(*Fixture*)

PROGRAM Fix108
	VAR_INPUT
		Enable_Prog: BOOL;
		Enable_Motion: BOOL;
		Discrete_In: udt_FixXX_Input_Image_20180202;
		Dry_Cycle: BOOL;
		Cell_In_Services: BOOL;
		Flash_Rate: BOOL;
		NodeLayout:udt_ECATNodeData_20221507;

	END_VAR

	VAR
(*Hardware Related Data Types*)
			(*Develop "Beckhoff Nodes"*)
			{attribute 'OPC.UA.DA':='1'}
			N00 AT %I*: udt_EP1111;
			{attribute 'OPC.UA.DA':='1'}
			N01 AT %I*: udt_EP1008_002_v2;
			{attribute 'OPC.UA.DA':='1'}
			N02 AT %I*: udt_EP1008_002_v2;
			{attribute 'OPC.UA.DA':='1'}
			N03 AT %I*: udt_EP1008_002_v2;
			{attribute 'OPC.UA.DA':='1'}
			N04 AT %I*: udt_EP1008_002_v2;
			{attribute 'OPC.UA.DA':='1'}
			N05 AT %I*: udt_EP1008_002_v2;
			{attribute 'OPC.UA.DA':='1'}
			N06 AT %I*: udt_EP1008_002_v2;
			{attribute 'OPC.UA.DA':='1'}
			N07 AT %I*: udt_EP1008_002_v2;
			{attribute 'OPC.UA.DA':='1'}
			N08 AT %I*: udt_EP1008_002_v2;
			{attribute 'OPC.UA.DA':='1'}
			N09 AT %I*: udt_EP1008_002_v2;
			{attribute 'OPC.UA.DA':='1'}
			N10 AT %I*: udt_EP1008_002_v2;
			{attribute 'OPC.UA.DA':='1'}
			N11 AT %I*: udt_EP1008_002_v2;
			{attribute 'OPC.UA.DA':='1'}
			N12 AT %I*: udt_EP1008_002_v2;
			{attribute 'OPC.UA.DA':='1'}
			N13 AT %I*: udt_EP1008_002_v2;
			{attribute 'OPC.UA.DA':='1'}
			N14 AT %I*: udt_EP1008_002_v2;
			{attribute 'OPC.UA.DA':='1'}
			N15 AT %I*: udt_EP1008_002_v2;
			{attribute 'OPC.UA.DA':='1'}
			N16 AT %I*: udt_EP1008_002_v2;
			{attribute 'OPC.UA.DA':='1'}
			N17 AT %I*: udt_EP1008_002_v2;
			{attribute 'OPC.UA.DA':='1'}
			N18 AT %I*: udt_EP1008_002_v2;
			{attribute 'OPC.UA.DA':='1'}
			N19 AT %I*: udt_EP1008_002_v2;
			{attribute 'OPC.UA.DA':='1'}
			N20 AT %I*: udt_EP1008_002_v2;
			{attribute 'OPC.UA.DA':='1'}
			N21 AT %I*: udt_EP1008_002_v2;
			{attribute 'OPC.UA.DA':='1'}
			N22 AT %I*: udt_EP1008_002_v2;
			{attribute 'OPC.UA.DA':='1'}
			N100 AT %Q*: udt_SMC_EX260_ValveBank;
			{attribute 'OPC.UA.DA':='1'}
			N100_STAT AT %I*:udt_SMC_EX260_Stat;
			{attribute 'OPC.UA.DA':='1'}
			N101 AT %Q*: udt_SMC_EX260_ValveBank;
			{attribute 'OPC.UA.DA':='1'}
			N101_STAT AT %I*:udt_SMC_EX260_Stat;
			{attribute 'OPC.UA.DA':='1'}
			N102 AT %Q*: udt_SMC_EX260_ValveBank;
			{attribute 'OPC.UA.DA':='1'}
			N102_STAT AT %I*:udt_SMC_EX260_Stat;

(* Nodes States*)
		NodeState: ARRAY[0..63] OF UINT;
		DiscreteNode_OK: BOOL;
(*Cable Break States*)
		ECatSlave_Cable_Breaks: ARRAY[0..1] OF DINT;
(*Standard Internal Variables*)
		(*Generic Sensor Variables*)
		All_Sensors_On: UINT;
		All_Sensors_Off: BOOL;
		All_Sensors_Off1: BOOL;
		All_Sensors_Off2: BOOL;
		(*Generic Position Variables*)
		Tool_At_Home: BOOL;
		Tool_At_Load: UINT;
		Tool_At_Weld: UINT;
		Tool_At_Rotate: UINT;
		Tool_At_Seal: UINT;
		Tool_At_Stud: UINT;
		Tool_At_Unload: UINT ;
		(*Grouping Of Items*)
		All_QAChecks_OK: BOOL;
		QAChecks_Failed: BOOL;
		(*General Internals*)
		In_Auto: BOOL;
		In_Manual: BOOL;

		Auto_Run: BOOL;
		Reset_All_Completes:BOOL;
		Load_Robots_Clear1: BOOL;
		Load_Robots_Clear2: BOOL;
		Load_Robots_Clear: BOOL;
		Load_Robots_WorkingOK1: BOOL;
		Load_Robots_WorkingOK2: BOOL;
		Load_Robots_Complete1: BOOL;
		Load_Robots_Complete2: BOOL;
		Load_Robots_PartInEOAT1: BOOL;
		Load_Robots_PartInEOAT2: BOOL;
		Load_Robots_UnclampEarly1: BOOL;
		Load_Robots_UnclampEarly2: BOOL;
		Seal_Robots_Clear: BOOL;
		Seal_Robots_WorkingOK: BOOL;
		Seal_Robots_UnclampEarly: BOOL;
		Seal_Robots_Complete: BOOL;
		Stud_Robots_Clear: BOOL;
		Stud_Robots_WorkingOK: BOOL;
		Stud_Robots_UnclampEarly: BOOL;
		Stud_Robots_Complete: BOOL;
		Weld_Robots_Clear: BOOL;
		Weld_Robots_WorkingOK: BOOL;
		Weld_Robots_UnclampEarly: BOOL;
		Weld_Robots_Complete: BOOL;
		Mig_Robots_Ready :BOOL;
		TurntableA_Clear: BOOL;
		TurntableB_Clear: BOOL;
		Turntable_Clear:BOOL;
		Turntable_WorkingOK: BOOL;
		TurntableA_Complete: BOOL;
		TurntableB_Complete: BOOL;
		Unload_Robots_Clear1: BOOL;
		Unload_Robots_WorkingOK1: BOOL;
		Unload_Robots_Complete1: BOOL;
		Unload_Robots_EOATEmpty1: BOOL;
		Unload_Robots_Clear2: BOOL;
		Unload_Robots_WorkingOK2: BOOL;
		Unload_Robots_Complete2: BOOL;
		Unload_Robots_EOATEmpty2: BOOL;
		Unload_Robots_Clear: BOOL;
		All_Robots_Clear: BOOL;

		Unload_Robot_Complete: BOOL;

		Start_Load_Robots1: BOOL;
		Start_Load_Robots2: BOOL;
		Start_Weld_Robots: BOOL;
		Start_Unload_Robots1: BOOL;
		Start_Unload_Robots2: BOOL;
		Start_Seal_Robots: BOOL;
		Start_Stud_Robots: BOOL;
		Start_TurntableA: BOOL;
		Start_TurntableB: BOOL;
		Load_Robots_Proceed1: BOOL;
		Load_Robots_Proceed2: BOOL;
		Weld_Robots_Proceed: BOOL;
		Seal_Robots_Proceed: BOOL;
		Stud_Robots_Proceed: BOOL;
		Unload_Robots_Proceed1: BOOL;
		Unload_Robots_Proceed2: BOOL;

		Prod_Inc: R_TRIG;
		Cycle_Time: TON;
		Cycle_Time_Pulse: R_TRIG;
		Load_Time: TON;
		Weld_Time: TON;
		Seal_Time: TON;
		Stud_Time: TON;
		Turn_Time: TON;
		Unload_Time: TON;
		Date_Stamp_TMR: TON;
		Date_StampHome_TMR: TON;
		CLFaulted: UDINT;
		PPFaulted: UDINT;
		Manual_Ind_HomePrompt: BOOL;
		Fixture_Allow_Model_Change: BOOL;

(*Non-Standard Variables*)

		(*FB Instances*)
		Clamp1FB: FB_Cylinder_Status;
		Clamp2FB: FB_Cylinder_Status;
		Clamp3FB: FB_Cylinder_Status;
		Clamp4FB: FB_Cylinder_Status;
		Clamp5FB: FB_Cylinder_Status;
		Clamp6FB: FB_Cylinder_Status;
		Clamp7FB: FB_Cylinder_Status;
		Clamp8FB: FB_Cylinder_Status;
		Clamp9FB: FB_Cylinder_Status;
		Clamp10FB: FB_Cylinder_Status;
		Clamp11FB: FB_Cylinder_Status;
		Clamp12FB: FB_Cylinder_Status;
		Clamp13FB: FB_Cylinder_Status;
		Clamp14FB: FB_Cylinder_Status;
		Clamp15FB: FB_Cylinder_Status;
		Clamp16FB: FB_Cylinder_Status;
		Clamp17FB: FB_Cylinder_Status;
		Clamp18FB: FB_Cylinder_Status;
		Clamp19FB: FB_Cylinder_Status;
		Clamp20FB: FB_Cylinder_Status;
		Clamp21FB: FB_Cylinder_Status;
		Clamp22FB: FB_Cylinder_Status;
		Clamp23FB: FB_Cylinder_Status;
		Clamp24FB: FB_Cylinder_Status;
		Cyl1FB: FB_TripleCylinder_20150625;
		Pin1FB: FB_Cylinder_Status;
		Pin2FB: FB_Cylinder_Status;
		Pin3FB: FB_Cylinder_Status;
		Pin4FB: FB_Cylinder_Status;
		Pin5FB: FB_Cylinder_Status;
		Pin6FB: FB_Cylinder_Status;
		Pin7FB: FB_Cylinder_Status;
		Pin8FB: FB_Cylinder_Status;
		Pin9FB: FB_Cylinder_Status;
		Pin10FB: FB_Cylinder_Status;
		Pin11FB: FB_Cylinder_Status;
		Pin12FB: FB_Cylinder_Status;
		Pin13FB: FB_Cylinder_Status;
		Pin14FB: FB_Cylinder_Status;
		Slide1FB: FB_Cylinder_Status;
		Slide2FB: FB_Cylinder_Status;
		Slide3FB: FB_Cylinder_Status;
		Slide4FB: FB_Cylinder_Status;
		Slide5FB: FB_Cylinder_Status;
		Slide6FB: FB_Cylinder_Status;
		Swing1FB: FB_Cylinder_Status;
		Swing2FB: FB_Cylinder_Status;
		Swing3FB: FB_Cylinder_Status;
		Swing4FB: FB_Cylinder_Status;
		Swing5FB: FB_Cylinder_Status;
		Swing6FB: FB_Cylinder_Status;
		QACheck1FB: FB_Cylinder_Status;
		QACheck2FB: FB_Cylinder_Status;
		CheckQA1FB: FB_GTAC_QAcheck_20150529;
		Part_Present1FB: FB_PP_Sensor;
		Part_Present2FB: FB_PP_Sensor;
		Part_Present3FB: FB_PP_Sensor;
		Part_Present4FB: FB_PP_Sensor;
		Part_Present5FB: FB_PP_Sensor;
		Part_Present6FB: FB_PP_Sensor;
		Part_Present7FB: FB_PP_Sensor;
		Part_Present8FB: FB_PP_Sensor;
		Part_Present9FB: FB_PP_Sensor;
		Part_Present10FB: FB_PP_Sensor;
		Part_Present11FB: FB_PP_Sensor;
		Part_Present12FB: FB_PP_Sensor;
		Part_Present13FB: FB_PP_Sensor;
		Part_Present14FB: FB_PP_Sensor;
		Part_Present15FB: FB_PP_Sensor;
		Part_Present16FB: FB_PP_Sensor;
		Part_Present17FB: FB_PP_Sensor;
		Part_Present18FB: FB_PP_Sensor;
		Part_Present19FB: FB_PP_Sensor;
		Part_Present20FB: FB_PP_Sensor;
		Part_Present21FB: FB_PP_Sensor;
		Part_Present22FB: FB_PP_Sensor;
		Part_Present23FB: FB_PP_Sensor;
		Part_Present24FB: FB_PP_Sensor;
		Part_Present25FB: FB_PP_Sensor;
		Part_Present26FB: FB_PP_Sensor;
		Part_Present27FB: FB_PP_Sensor;
		Part_Present28FB: FB_PP_Sensor;
		Part_Present29FB: FB_PP_Sensor;
		Part_Present30FB: FB_PP_Sensor;
		Part_Present31FB: FB_PP_Sensor;
		Part_Present32FB: FB_PP_Sensor;
		Part_Present33FB: FB_PP_Sensor;
		Part_Present34FB: FB_PP_Sensor;
		Part_Present35FB: FB_PP_Sensor;
		Part_Present36FB: FB_PP_Sensor;
		Part_Present37FB: FB_PP_Sensor;
		Part_Present38FB: FB_PP_Sensor;
		Part_Present39FB: FB_PP_Sensor;
		Part_Present40FB: FB_PP_Sensor;
		Tape_Present1FB: FB_PP_Sensor;

		(*Valve FBs*)
		Valve1FB: FB_GTAC_Valve_20170704;
		Valve2FB: FB_GTAC_Valve_20170704;
		Valve3FB: FB_GTAC_Valve_20170704;
		Valve4FB: FB_GTAC_Valve_20170704;
		Valve5FB: FB_GTAC_Valve_20170704;
		Valve6FB: FB_GTAC_Valve_20170704;
		Valve7FB: FB_GTAC_Valve_20170704;
		Valve8FB: FB_GTAC_Valve_20170704;
		Valve9FB: FB_GTAC_Valve_20170704;
		Valve10FB: FB_GTAC_Valve_20170704;
		Valve11FB: FB_GTAC_Valve_20170704;
		Valve12FB: FB_GTAC_Valve_20170704;
		Valve13FB: FB_GTAC_Valve_20170704;
		Valve14FB: FB_GTAC_Valve_20170704;
		Valve15FB: FB_GTAC_Valve_20170704;
		Valve16FB: FB_GTAC_Valve_20170704;
		Valve17FB: FB_GTAC_Valve_20170704;
		Valve18FB: FB_GTAC_Valve_20170704;
		Valve19FB: FB_GTAC_Valve_20170704;
		Valve20FB: FB_GTAC_Valve_20170704;
		Valve21FB: FB_GTAC_Valve_20170704;
		Valve22FB: FB_GTAC_Valve_20170704;
		Valve23FB: FB_GTAC_Valve_20170704;
		Valve24FB: FB_GTAC_Valve_20170704;
		Valve25FB: FB_GTAC_Valve_20170704;
		Valve26FB: FB_GTAC_Valve_20170704;
		Valve27FB: FB_GTAC_Valve_20170704;
		Valve28FB: FB_GTAC_Valve_20170704;
		Valve29FB: FB_GTAC_Valve_20170704;
		Valve30FB: FB_GTAC_Valve_20170704;
		Valve31FB: FB_GTAC_Valve_20170704;
		Valve32FB: FB_GTAC_Valve_20170704;
		Valve33FB: FB_GTAC_Valve_20170704;
		Valve34FB: FB_GTAC_Valve_20170704;
		Valve35FB: FB_GTAC_Valve_20170704;
		Valve36FB: FB_GTAC_Valve_20170704;
		Valve37FB: FB_GTAC_Valve_20170704;
		Valve38FB: FB_GTAC_Valve_20170704;
		Valve39FB: FB_GTAC_Valve_20170704;
		Valve40FB: FB_GTAC_Valve_20170704;
		Valve41FB: FB_GTAC_Valve_20170704;
		Valve42FB: FB_GTAC_Valve_20170704;
		Valve43FB: FB_GTAC_Valve_20170704;
		Valve44FB: FB_GTAC_Valve_20170704;
		Valve45FB: FB_GTAC_Valve_20170704;
		Valve46FB: FB_GTAC_Valve_20170704;
		Valve47FB: FB_GTAC_Valve_20170704;
		Valve48FB: FB_GTAC_Valve_20170704;

		(*Tool Positions*)
			(*Add User Indivdual Position Variables Here*)
			Clamp1ADVD: BOOL;
			Clamp1RETD: BOOL;
			Clamp2ADVD: BOOL;
			Clamp2RETD: BOOL;
			Clamp3ADVD: BOOL;
			Clamp3RETD: BOOL;
			Clamp4ADVD: BOOL;
			Clamp4RETD: BOOL;
			Clamp5ADVD: BOOL;
			Clamp5RETD: BOOL;
			Clamp6ADVD: BOOL;
			Clamp6RETD: BOOL;
			Clamp7ADVD: BOOL;
			Clamp7RETD: BOOL;
			Clamp8ADVD: BOOL;
			Clamp8RETD: BOOL;
			Clamp9ADVD: BOOL;
			Clamp9RETD: BOOL;
			Clamp10ADVD: BOOL;
			Clamp10RETD: BOOL;
			Clamp11ADVD: BOOL;
			Clamp11RETD: BOOL;
			Clamp12ADVD: BOOL;
			Clamp12RETD: BOOL;
			Clamp13ADVD: BOOL;
			Clamp13RETD: BOOL;
			Clamp14ADVD: BOOL;
			Clamp14RETD: BOOL;
			Clamp15ADVD: BOOL;
			Clamp15RETD: BOOL;
			Clamp16ADVD: BOOL;
			Clamp16RETD: BOOL;
			Clamp17ADVD: BOOL;
			Clamp17RETD: BOOL;
			Clamp18ADVD: BOOL;
			Clamp18RETD: BOOL;
			Clamp19ADVD: BOOL;
			Clamp19RETD: BOOL;
			Clamp20ADVD: BOOL;
			Clamp20RETD: BOOL;
			Clamp21ADVD: BOOL;
			Clamp21RETD: BOOL;
			Clamp22ADVD: BOOL;
			Clamp22RETD: BOOL;
			Clamp23ADVD: BOOL;
			Clamp23RETD: BOOL;
			Clamp24ADVD: BOOL;
			Clamp24RETD: BOOL;
			Cyl1ADVD: BOOL;
			Cyl1MID: BOOL;
			Cyl1RETD: BOOL;
			Pin1ADVD: BOOL;
			Pin1RETD: BOOL;
			Pin2ADVD: BOOL;
			Pin2RETD: BOOL;
			Pin3ADVD: BOOL;
			Pin3RETD: BOOL;
			Pin4ADVD: BOOL;
			Pin4RETD: BOOL;
			Pin5ADVD: BOOL;
			Pin5RETD: BOOL;
			Pin6ADVD: BOOL;
			Pin6RETD: BOOL;
			Pin7ADVD: BOOL;
			Pin7RETD: BOOL;
			Pin8ADVD: BOOL;
			Pin8RETD: BOOL;
			Pin9ADVD: BOOL;
			Pin9RETD: BOOL;
			Pin10ADVD: BOOL;
			Pin10RETD: BOOL;
			Pin11ADVD: BOOL;
			Pin11RETD: BOOL;
			Pin12ADVD: BOOL;
			Pin12RETD: BOOL;
			Pin13ADVD: BOOL;
			Pin13RETD: BOOL;
			Pin14ADVD: BOOL;
			Pin14RETD: BOOL;
			Slide1ADVD: BOOL;
			Slide1RETD: BOOL;
			Slide2ADVD: BOOL;
			Slide2RETD: BOOL;
			Slide3ADVD: BOOL;
			Slide3RETD: BOOL;
			Slide4ADVD: BOOL;
			Slide4RETD: BOOL;
			Slide5ADVD: BOOL;
			Slide5RETD: BOOL;
			Slide6ADVD: BOOL;
			Slide6RETD: BOOL;
			Swing1ADVD: BOOL;
			Swing1RETD: BOOL;
			Swing2ADVD: BOOL;
			Swing2RETD: BOOL;
			Swing3ADVD: BOOL;
			Swing3RETD: BOOL;
			Swing4ADVD: BOOL;
			Swing4RETD: BOOL;
			Swing5ADVD: BOOL;
			Swing5RETD: BOOL;
			Swing6ADVD: BOOL;
			Swing6RETD: BOOL;
			QACheck1ADVD: BOOL;
			QACheck1RETD: BOOL;
			QACheck2ADVD: BOOL;
			QACheck2RETD: BOOL;

		(*Part Present Sensors*)
			(*Main Body Present*)
			Part_Present1: BOOL;
			Part_Present2: BOOL;
			Part_Present3: BOOL;
			Part_Present4: BOOL;
			Part_Present5: BOOL;
			Part_Present6: BOOL;
			Part_Present7: BOOL;
			Part_Present8: BOOL;
			Part_Present9: BOOL;
			Part_Present10: BOOL;
			Part_Present11: BOOL;
			Part_Present12: BOOL;
			Part_Present13: BOOL;
			Part_Present14: BOOL;
			Part_Present15: BOOL;
			Part_Present16: BOOL;
			Part_Present17: BOOL;
			Part_Present18: BOOL;
			Part_Present19: BOOL;
			Part_Present20: BOOL;
			Part_Present21: BOOL;
			Part_Present22: BOOL;
			Part_Present23: BOOL;
			Part_Present24: BOOL;
			Part_Present25: BOOL;
			Part_Present26: BOOL;
			Part_Present27: BOOL;
			Part_Present28: BOOL;
			Part_Present29: BOOL;
			Part_Present30: BOOL;
			Part_Present31: BOOL;
			Part_Present32: BOOL;
			Part_Present33: BOOL;
			Part_Present34: BOOL;
			Part_Present35: BOOL;
			Part_Present36: BOOL;
			Part_Present37: BOOL;
			Part_Present38: BOOL;
			Part_Present39: BOOL;
			Part_Present40: BOOL;
			Tape_Present1: BOOL;

		(*Motion Sequence Variables*)
			Clamp_Step: UINT;
			Repo1_Step: UINT;
			Repo2_Step: UINT;
			Repo3_Step: UINT;
			Repo4_Step: UINT;
			Unclamp_Step: UINT;

		(*Custom Application Variables*)
			Weld_Curtain_Bypass: BOOL;
			Vacuum_Bypass: BOOL;
			Sealer_Bypass: BOOL;
			Stud_Bypass: BOOL;

END_VAR

	(*data that needs to be retained in the event of a power cycle*)
	VAR PERSISTENT

		Load_Complete1: BOOL;
		Load_Complete2: BOOL;
		Load_Complete: BOOL;
		Stud_Complete: BOOL;
		Welding_Complete: BOOL;
		Sealing_Complete: BOOL;
		Unload_Complete: BOOL;
		TurnA_Complete: BOOL;
		TurnB_Complete: BOOL;
		Cycle_Complete: BOOL;
		Eject_Complete: BOOL;
		VacCheck_Complete: BOOL;
		Date_Stamp_Complete: BOOL;
		Load_Seq01: FB_GTAC_Load_Seq_20230302;
		Production_Count:INT;
		Repo_REQS: UINT;
		(*Allow_Load_PreCall: BOOL;
		Allow_Weld_PreCall: BOOL;
		Allow_Unload_PreCall: BOOL;*)
		(*All_SubPP_Off: BOOL;*)
		Production_Report: FB_Production_Report_20221007;

	END_VAR

	VAR_OUTPUT

		Prog_Ok: BOOL;
		Discrete_Image: udt_FixXX_Output_Image_20220715;
		In_Auto_Mode: BOOL;
		In_Manual_Mode: BOOL;
		Manual_Indicators1: DINT;
		Manual_Indicators2: DINT;
		Manual_Indicators3: DINT;
		At_Home: BOOL;
		Ready_To_Load: BOOL;
		Red_Lamp_Req: BOOL;
		Status: UINT;
		CLFaults1:UDINT;
		CLFaults2:UDINT;
		CLFaults3:UDINT;
		CLFaults4:UDINT;
		PPFaults: UDINT;
		PPFaults1: UDINT;
		PPFaults2: UDINT;
		Prod_Count_Out: INT;
		Cycle_Time_Out: TIME;
		PrevCycle_Time_Out: TIME;
		Load_Time_Out: TIME;
		Weld_Time_Out: TIME;
		Seal_Time_Out: TIME;
		Stud_Time_Out: TIME;
		Turn_Time_Out: TIME;
		Unload_Time_Out: TIME;
		Model_ID: UINT;
		TurntableA_At_Robot: BOOL;
		TurntableB_At_Robot: BOOL;
		Tool_Call_ForLoadRobots1: BOOL;
		Tool_Call_ForLoadRobots2: BOOL;
		Tool_Call_ForSealRobots: BOOL;
		Tool_Call_ForStudRobots: BOOL;
		Tool_Call_ForWeldRobots: BOOL;
		Tool_Call_ForSweepA: BOOL;
		Tool_Call_ForSweepB: BOOL;
		Tool_Call_ForUnloadRobots1: BOOL;
		Tool_Call_ForUnloadRobots2: BOOL;
		Robots_Clear_ToProceed: BOOL;
		Task_ID: UINT;
		Fix_ID: UINT;
		Load_Complete1_Ack: BOOL;
		Load_Complete2_Ack: BOOL;
		Seal_Complete_Ack: BOOL;
		Stud_Complete_Ack: BOOL;
		Weld_Complete_Ack: BOOL;
		TurnA_Complete_Ack: BOOL;
		TurnB_Complete_Ack: BOOL;
		Unload_Complete1_Ack: BOOL;
		Unload_Complete2_Ack: BOOL;
		Repo_Ack: UINT;
	END_VAR

	(*Set FB_OK to True*)
	Prog_OK:= TRUE;


	(*Set conditions to allow model change*)
	Fixture_Allow_Model_Change:= (In_Manual AND Tool_At_Home AND All_Sensors_Off AND All_Robots_Clear)
							OR (Model_ID=0);



(*$$$$$$$$$$$$$$$$$$$$$$$$$$$$$$$$$$$$$$$$$$$$ Fixture Bypasses $$$$$$$$$$$$$$$$$$$$$$$$$$$$$$$$$$$$$$$$$$$$$$$$$$$$*)
	Weld_Curtain_Bypass:= Discrete_In.Bypass_REQS.0;
	Vacuum_Bypass:= Discrete_In.Bypass_REQS.1;
	Stud_Bypass:= Discrete_In.Bypass_REQS.2;
	Sealer_Bypass:= MAIN.SL01.Disp1_Bypass;


(*$$$$$$$$$$$$$$$$$$$$$$$$$$$$$$$$$$$$$$$$$$$$ Gather Status Of Hardware $$$$$$$$$$$$$$$$$$$$$$$$$$$$$$$$$$$$$$$$$$$$$$$$$$$$*)
	(*Check on Status of Hardware*)
	Hardware();

(*$$$$$$$$$$$$$$$$$$$$$$$$$$$$$$$$$$$$$$$$$$$$$ Gather Standard Inputs $$$$$$$$$$$$$$$$$$$$$$$$$$$$$$$$$$$$$$$$$$$$$$$$$$$$$$$$$*)

(*Clamp/Cylinder Inputs*)
	Cylinders();

(*Part Present Inputs*)
	Proxies();

(*$$$$$$$$$$$$$$$$$$$$$$$$$$$$$$$$$$$$$$$$$$$ Qaulity Checking Routines $$$$$$$$$$$$$$$$$$$$$$$$$$$$$$$$$$$$$$$$$$$$$$$$$$$$$$$$$*)

	(*QA Checks*)
		CheckQA1FB(
			Start_QAcheck:= Auto_Run AND Enable_Motion AND Tool_At_Load.3,
			QAcheck_Reset:= Cycle_Complete OR (In_Manual AND Discrete_In.Go_Home AND All_Sensors_Off),
			QAcheck_Retry:= In_From_ICxx.QA_Reset.0,
			QAcheck_Release:= In_From_ICxx.QA_Reset.1,
			QAcheck_Adv_In:= QACheck1ADVD AND QACheck2ADVD,
			QAcheck_Ret_In:= QACheck1RETD AND QACheck2RETD,
			User_Dry_Cycle:= Dry_Cycle,
			QAcheck_OK_Delay:= T#0.75s,
			QAcheck_Fault_Delay:= T#3.0s,
			QAcheck_OK=> All_QAChecks_OK,
			QAcheck_Failed=> QAChecks_Failed);



(*$$$$$$$$$$$$$$$$$$$$$$$$$$$$$$$$$$$$$$$$$$$$$$$$ Internal Code $$$$$$$$$$$$$$$$$$$$$$$$$$$$$$$$$$$$$$$$$$$$$$$$$$$$$$$$$$$$$$$$$$$$*)
(*Auto / Manual Mode Code*)
	IF Discrete_In.Mode_Select.0 AND NOT Discrete_In.Mode_Select.1
		THEN
			In_Auto:= TRUE;
			In_Auto_Mode:= TRUE;
	END_IF;
	IF NOT Discrete_In.Mode_Select.0 AND Discrete_In.Mode_Select.1
		THEN
			In_Auto:= FALSE;
			In_Auto_Mode:= FALSE;
	END_IF;
	In_Manual:= NOT In_Auto;
	In_Manual_Mode:= In_Manual;

(*--------------------------------------------------------------------------------Tool Positions---------------------------------------------------------------*)
	Tool_States();

(*----------------------------------------------------Part Present Sensor Input Patterns----------------------------------------------------------------*)
	All_Sensors();


(*>>>>>>>>>>>>>>>>>>>>>>>>>>>>>>>>>>>>>>>>>> Auto Run Cycle >>>>>>>>>>>>>>>>>>>>>>>>>>>>>>>>>>>>>>>*)
(*+++++++++++THIS AREA IS CUSTOM PER INSTALLATION AND WILL HAVE TO BE MODIFIED PER +++++++++++++*)
(*+++++++++++THIS AREA IS CUSTOM PER INSTALLATION AND WILL HAVE TO BE MODIFIED PER +++++++++++++*)
	(*Control of Auto_Run*)
	Auto_Run:= Enable_Motion AND In_Auto AND Model_ID<>0 AND NOT Cycle_Complete;

	(*Auto Run Enables All Other Auto Cycle Code*)
	IF Auto_Run
		THEN

			IF (NOT Load_Complete1 OR (Load_Robots_UnclampEarly1 AND All_Sensors_On.1))
				AND Load_Robots_Clear2 AND Stud_Robots_Clear AND Seal_Robots_Clear
				AND Weld_Robots_Clear AND TurnTable_Clear AND Unload_Robots_Clear
				AND TurnTableA_At_Robot
				THEN
					(*Start 1st Load Robots*)
					Start_Load_Robots1:= ((Tool_At_Load.0 AND All_Sensors_Off AND NOT Repo_Reqs.0 AND Load_Robots_PartInEOAT1)
									OR (Tool_At_Load.1 AND All_Sensors_On.4 AND Repo_Reqs.0))
									OR Load_Robots_WorkingOK1;
					(*Allow 1st Load Robots To Proceed*)
					Load_Robots_Proceed1:= Tool_At_Load.0 AND All_Sensors_Off AND Load_Robots_PartInEOAT1;
			ELSE
					Start_Load_Robots1:= FALSE;
					Load_Robots_Proceed1:= FALSE;
			END_IF;


			IF (NOT Load_Complete2 OR (Load_Robots_UnclampEarly2 AND All_Sensors_On.2))
				AND Load_Robots_Clear1 AND Stud_Robots_Clear AND Seal_Robots_Clear
				AND Weld_Robots_Clear AND TurnTable_Clear AND Unload_Robots_Clear
				AND TurnTableA_At_Robot
				THEN
					(*Start 2nd Load Robots*)
					Start_Load_Robots2:= ((Tool_At_Load.1 AND All_Sensors_Off AND NOT Repo_Reqs.0 AND Load_Robots_PartInEOAT2)
									OR (Tool_At_Load.1 AND All_Sensors_On.4 AND Repo_Reqs.0))
									OR Load_Robots_WorkingOK2;
					(*Allow 2nd Load Robots To Proceed*)
					Load_Robots_Proceed2:= Tool_At_Load.1 AND All_Sensors_Off AND Load_Robots_PartInEOAT2;
			ELSE
					Start_Load_Robots2:= FALSE;
					Load_Robots_Proceed2:= FALSE;
			END_IF;


			IF NOT Sealer_Bypass AND Load_Complete AND NOT Sealing_Complete
				AND Load_Robots_Clear AND Stud_Robots_Clear AND  Weld_Robots_Clear AND TurnTable_Clear AND Unload_Robots_Clear
				AND TurnTableA_At_Robot
				THEN
					(*Start Seal Robots*)
					Start_Seal_Robots:= ((Tool_At_Seal.0 AND All_Sensors_On.3 AND NOT Repo_Reqs.1 AND NOT MAIN.SL01.Disp1_Faulted AND MAIN.SL01.Disp1_Ready)
									OR (Tool_At_Seal.1 AND All_Sensors_On.4 AND Repo_Reqs.1))
									OR Seal_Robots_WorkingOK;
					(*Allow Seal Robots To Proceed*)
					Seal_Robots_Proceed:= Tool_At_Seal.0 AND All_Sensors_On.3;
			ELSE
					Start_Seal_Robots:= FALSE;
					Seal_Robots_Proceed:= FALSE;
			END_IF;


			IF NOT Stud_Bypass AND Load_Complete AND NOT Stud_Complete AND NOT Welding_Complete
				AND Load_Robots_Clear AND Seal_Robots_Clear AND  Weld_Robots_Clear AND TurnTable_Clear AND Unload_Robots_Clear
				AND TurnTableA_At_Robot
				THEN
					(*Start Stud Robots*)
					Start_Stud_Robots:= ((Tool_At_Stud.0 AND All_Sensors_On.3 AND NOT Repo_Reqs.2)
									OR (Tool_At_Stud.1 AND All_Sensors_On.4 AND Repo_Reqs.2))
									OR Stud_Robots_WorkingOK;
					(*Allow Stud Robots To Proceed*)
					Stud_Robots_Proceed:= Tool_At_Stud.0 AND All_Sensors_On.3;
			ELSE
					Start_Stud_Robots:= FALSE;
					Stud_Robots_Proceed:= FALSE;
			END_IF;


                             IF  NOT TurnA_Complete AND Load_Complete AND NOT Welding_Complete AND NOT Unload_Complete
				 AND Load_Robots_Clear AND Seal_Robots_Clear AND Stud_Robots_Clear AND  Weld_Robots_Clear AND Unload_Robots_Clear
				AND (NOT TurntableA_At_Robot OR TurnTable_WorkingOK)
				THEN
					(*Start Turntable SweepA (Fix01 to the Robot)*)
					Start_TurntableA:= ((Tool_At_Rotate.0 AND All_Sensors_On.3)
									OR (All_Sensors_Off AND Tool_At_Home))
									OR TurnTable_WorkingOK;
			ELSE
					Start_TurntableA:= FALSE;
			END_IF;


			IF NOT TurnB_Complete AND Welding_Complete AND NOT Unload_Complete AND (Sealing_Complete OR Sealer_Bypass) AND (Stud_Complete OR Stud_Bypass)
				AND Load_Robots_Clear AND Seal_Robots_Clear AND Stud_Robots_Clear AND Weld_Robots_Clear  AND Unload_Robots_Clear
				AND (NOT TurntableB_At_Robot OR TurnTable_WorkingOK)
				THEN
					(*Start Turntable SweepB (Fix01 to the Operator)*)
					Start_TurntableB:= TRUE;
                             ELSIF All_Sensors_Off AND NOT TurnB_Complete AND Weld_Robots_Clear AND Load_Robots_Clear AND Unload_Robots_Clear
				AND (NOT TurntableB_At_Robot OR TurnTable_WorkingOK)
			THEN
					Start_TurntableB:= All_Sensors_Off;
                             ELSE
					Start_TurntableB:= FALSE;
                             END_IF;


			IF Load_Complete AND NOT Welding_Complete AND (Sealing_Complete OR Sealer_Bypass) AND (Stud_Complete OR Stud_Bypass) AND NOT Unload_Complete
				AND Load_Robots_Clear AND Seal_Robots_Clear AND Stud_Robots_Clear AND TurnTable_Clear AND Unload_Robots_Clear
				AND TurnTableA_At_Robot AND Mig_Robots_Ready 
				THEN
					(*Start Weld Robots*)
					Start_Weld_Robots:=((Tool_At_Weld.0 AND NOT Repo_Reqs.3 AND NOT Repo_Reqs.4 AND NOT Repo_Reqs.5 AND All_Sensors_On.3)
										OR (Tool_At_Weld.1 AND Repo_Reqs.3 AND All_Sensors_On.3)
										OR (Tool_At_Weld.2 AND Repo_Reqs.4 AND All_Sensors_On.4)
										OR (Tool_At_Weld.3 AND Repo_Reqs.5 AND All_Sensors_On.5)
										OR (Tool_At_Unload.0 AND Weld_Robots_UnclampEarly))
										OR Weld_Robots_WorkingOK;
					(*Allow Weld Robots To Proceed*)
					Weld_Robots_Proceed:= Load_Complete AND Tool_At_Weld.0 AND All_Sensors_On.3;
			ELSE
					Start_Weld_Robots:= FALSE;
					Weld_Robots_Proceed:= FALSE;
			END_IF;


			IF Welding_Complete  AND (Sealing_Complete OR Sealer_Bypass) AND (Stud_Complete OR Stud_Bypass) AND NOT Unload_Complete
				AND Load_Robots_Clear AND Seal_Robots_Clear AND Stud_Robots_Clear AND TurnTable_Clear AND Unload_Robots_Clear2
				AND TurnTableA_At_Robot
				THEN
					(*Start Unload Robots*)
					Start_Unload_Robots1:=((((Tool_At_Unload.0 AND NOT Repo_Reqs.6 AND NOT Repo_Reqs.7 AND All_Sensors_On.8)
										OR (Tool_At_Unload.1 AND Repo_Reqs.6)
										OR (Tool_At_Unload.2 AND Repo_Reqs.7))
										AND (All_Sensors_On.8 AND Unload_Robots_EOATEmpty1))
										OR (NOT Unload_Robots_Clear1 AND NOT Unload_Robots_EOATEmpty1))
										OR Unload_Robots_WorkingOK1;
					(*Allow Unload Robots To Proceed*)
					Unload_Robots_Proceed1:= Welding_Complete AND Tool_At_Unload.0 AND All_Sensors_On.8 AND Unload_Robots_EOATEmpty1;
			ELSE
					Start_Unload_Robots1:= FALSE;
					Unload_Robots_Proceed1:= FALSE;
			END_IF;


			IF Welding_Complete  AND (Sealing_Complete OR Sealer_Bypass) AND (Stud_Complete OR Stud_Bypass) AND NOT Unload_Complete
				AND Load_Robots_Clear AND Seal_Robots_Clear AND Stud_Robots_Clear AND TurnTable_Clear AND Unload_Robots_Clear1
				AND TurnTableA_At_Robot
				THEN
					(*Start Unload Robots*)
					Start_Unload_Robots2:=((((Tool_At_Unload.0 AND NOT Repo_Reqs.6 AND NOT Repo_Reqs.7 AND All_Sensors_On.8)
										OR (Tool_At_Unload.1 AND Repo_Reqs.6)
										OR (Tool_At_Unload.2 AND Repo_Reqs.7))
										AND (All_Sensors_On.8 AND Unload_Robots_EOATEmpty2))
										OR (NOT Unload_Robots_Clear2 AND NOT Unload_Robots_EOATEmpty2))
										OR Unload_Robots_WorkingOK2;
					(*Allow Unload Robots To Proceed*)
					Unload_Robots_Proceed2:= Welding_Complete AND Tool_At_Unload.0 AND All_Sensors_On.8 AND Unload_Robots_EOATEmpty2;
			ELSE
					Start_Unload_Robots2:= FALSE;
					Unload_Robots_Proceed2:= FALSE;
			END_IF;


	ELSE
		Start_Load_Robots1:= FALSE;
		Start_Load_Robots2:= FALSE;
		Start_Seal_Robots:= FALSE;
		Start_Stud_Robots:= FALSE;
		Start_TurntableA:= FALSE;
		Start_TurntableB:= FALSE;
		Start_Weld_Robots:= FALSE;
		Start_Unload_Robots1:= FALSE;
		Start_Unload_Robots2:= FALSE;
		Load_Robots_Proceed1:=FALSE;
		Load_Robots_Proceed2:=FALSE;
		Seal_Robots_Proceed:=FALSE;
		Weld_Robots_Proceed:=FALSE;
		Unload_Robots_Proceed1:=FALSE;
		Unload_Robots_Proceed2:=FALSE;
	END_IF;




(*---------------------------------------------------------------Completes----------------------------------------------------*)
	(*1st Load Complete*)
	IF NOT Dry_Cycle
		THEN
		Load_Complete1:=  All_Sensors_On.1;
	ELSIF Dry_Cycle
		THEN
		IF Tool_At_Home AND Enable_Motion AND All_Sensors_Off
			THEN
			Load_Complete1:= TRUE;
		END_IF;
	END_IF;
	(*2nd Load Complete*)
	IF NOT Dry_Cycle
		THEN
		Load_Complete2:=  All_Sensors_On.2;
	ELSIF Dry_Cycle
		THEN
		IF Tool_At_Home AND Enable_Motion AND All_Sensors_Off
			THEN
			Load_Complete2:= TRUE;
		END_IF;
	END_IF;
	(*All Load Complete*)
	IF NOT Dry_Cycle
		THEN
		Load_Complete:= (All_Sensors_On.2
					OR (All_Sensors_On.3 AND Tool_At_Weld.0)
					OR (Repo_Reqs.0 AND All_Sensors_On.4)
					OR (Repo_Reqs.1 AND All_Sensors_On.5)
					OR (Repo_Reqs.2 AND All_Sensors_On.6))
					OR Weld_Robots_WorkingOK OR Welding_Complete;
	ELSIF Dry_Cycle
		THEN
		IF Load_Complete1 AND Load_Complete2 AND All_Sensors_Off
			THEN
			Load_Complete:= TRUE;
		END_IF;
	END_IF;

	(*Welding Complete*)
	IF Weld_Robots_Complete
		THEN
		Welding_Complete:= TRUE;
	END_IF;

	(*Unload Complete*)
	IF NOT Dry_Cycle
		THEN
			IF (Unload_Robots_Complete1 OR Unload_Robots_Complete2 OR (All_Sensors_Off AND Unload_Robots_Clear)) AND Welding_Complete
				THEN
				Unload_Complete:= TRUE;
			END_IF;
	ELSIF Dry_Cycle
		THEN
			IF (Unload_Robots_Complete1 OR Unload_Robots_Complete2 OR (All_Sensors_Off AND Unload_Robots_Clear)) AND Welding_Complete
				THEN
				Unload_Complete:= TRUE;
			END_IF;
	END_IF;
(*!!!!!!!!!!!!!!!!!!!!!!!!!!!!!!!!!!!!!!!!!!!!!!!!!!!!!!!!!!!!!!!!!!!!!!!!!!!!!!!!!!!!!!!!!!!!!!!!! Cycle Complete !!!!!!!!!!!!!!!!!!!!!!!!!!!!!!!!!!!!!!!!!!!!!!!!!!!!!!!!!!!!!!!!!!!!!!!!!!!!!!!!!!!!!!!!!!*)
	(*Set Cycle Complete*)
	IF Auto_Run AND Load_Complete AND Welding_Complete AND Unload_Complete AND All_Robots_Clear
		THEN Cycle_Complete:= TRUE;
	END_IF;
	(*Reset All Completes*)
	IF Load_Robots_Clear AND Weld_Robots_Clear AND Unload_Robots_Clear AND NOT Unload_Robots_Complete1 AND NOT Unload_Robots_Complete2
		THEN
			IF In_Manual AND Discrete_In.Go_Home AND All_Sensors_Off
				THEN
					Reset_All_Completes:= TRUE;
			ELSIF NOT Dry_Cycle AND Cycle_Complete AND NOT Enable_Motion AND Tool_At_Home AND All_Sensors_Off
				THEN
					Reset_All_Completes:= TRUE;
			ELSIF Dry_Cycle AND Cycle_Complete AND Tool_At_Home AND All_Sensors_Off
				THEN
					Reset_All_Completes:=TRUE;
			ELSE
					Reset_All_Completes:= FALSE;
			END_IF;
	END_IF;
	(*Perform Actual Reset*)
		IF Reset_All_Completes
			THEN
				Cycle_Complete:= FALSE;
				Load_Complete1:= FALSE;
				Load_Complete2:= FALSE;
				Load_Complete:= FALSE;
				Sealing_Complete:= FALSE;
				Stud_Complete:= FALSE;
				Welding_Complete:= FALSE;
				Date_Stamp_Complete:= FALSE;
				VacCheck_Complete:= FALSE;
				Unload_Complete:=FALSE;
				Eject_Complete:= FALSE;
				Load_Robots_UnclampEarly1:= FALSE;
				Load_Robots_UnclampEarly2:= FALSE;
				Seal_Robots_UnclampEarly:= FALSE;
				Stud_Robots_UnclampEarly:= FALSE;
				Weld_Robots_UnclampEarly:= FALSE;
				Repo_Reqs:= 0;
				Reset_All_Completes:= FALSE;

		END_IF;

(*---------------------------------------------------------------------------- Call Various Actions ----------------------------------------------------------------------------------------------------*)
	(*Poduction Counters and Report*)
	Production();

	(*Register Robot(s) to Fixture*)
	Robot_Registration();

	(*Setup Fix ID and Model Data*)
	Task_Fix_Model_IDs();

	(*Generate Status Banner and Fault Flags*)
	Status_and_Faults();

	(*Tool Clamp / Unclamp Sequencing and Reposition Handling*)
	Tool_VBSeq_Repos();

	(*Transfer Object Image Data to UI Section*)
	Xfer_To_UI();


(*-----------------------------------------------------------------------------------------Transfer Valve Outputs --------------------------------------------------------------------------------*)
	(*Move "Manual_Home_Prompt" as required for home prompting*)
		Manual_Ind_HomePrompt:= Flash_Rate AND In_Manual AND Discrete_In.Go_Home AND NOT Tool_At_Home;

	(*Call each valve bank*)
	ValveBank1();
	(*ValveBank2();
	ValveBank3(); *)

ACTION All_Sensors:


(*+++++++++++THIS AREA IS CUSTOM PER INSTALLATION AND WILL HAVE TO BE MODIFIED PER +++++++++++++*)
(*+++++++++++THIS AREA IS CUSTOM PER INSTALLATION AND WILL HAVE TO BE MODIFIED PER +++++++++++++*)
(*+++++++++++THIS AREA IS CUSTOM PER INSTALLATION AND WILL HAVE TO BE MODIFIED PER +++++++++++++*)



(**************************************************************************All Sensors Off******************************************************************************)
(**************************************************************************All Sensors Off******************************************************************************)
(**************************************************************************All Sensors Off******************************************************************************)

	(*All Sensors Required Off*)
	All_Sensors_Off:= NOT Part_Present1 AND NOT Part_Present2 AND NOT  Part_Present3
			AND NOT Part_Present4 AND NOT Part_Present5 AND NOT Part_Present6
			AND NOT Part_Present7 AND NOT Part_Present8 AND NOT Part_Present9
			AND NOT Part_Present10 AND NOT Part_Present11 AND NOT Part_Present12
			AND NOT Part_Present13 AND NOT Part_Present14 AND NOT Part_Present15
			AND NOT Part_Present16 AND NOT Part_Present17 AND NOT Part_Present18
			AND NOT Part_Present19 AND NOT Part_Present20 AND NOT Part_Present21
			AND NOT Part_Present22 AND NOT Part_Present23 AND NOT Part_Present24
			AND NOT Part_Present25 AND NOT Part_Present26 AND NOT Part_Present27
			AND NOT Part_Present28 AND NOT Part_Present29 AND NOT Part_Present30
			AND NOT Part_Present31 AND NOT Part_Present32 AND NOT Part_Present33
			AND NOT Part_Present34 AND NOT Part_Present35 AND NOT Part_Present36
			AND NOT Part_Present37 AND NOT Part_Present38 AND NOT Part_Present39
			AND NOT Part_Present40;

	(*All Sensors Required Off - Used for sub fixtures where the part has to move from one stage to the next*)
	All_Sensors_Off1:= NOT Part_Present1 AND NOT Part_Present2 AND NOT  Part_Present3
			AND NOT Part_Present4 AND NOT Part_Present5 AND NOT Part_Present6
			AND NOT Part_Present7 AND NOT Part_Present8 AND NOT Part_Present9
			AND NOT Part_Present10 AND NOT Part_Present11 AND NOT Part_Present12
			AND NOT Part_Present13 AND NOT Part_Present14 AND NOT Part_Present15
			AND NOT Part_Present16 AND NOT Part_Present17 AND NOT Part_Present18
			AND NOT Part_Present19 AND NOT Part_Present20 AND NOT Part_Present21
			AND NOT Part_Present22 AND NOT Part_Present23 AND NOT Part_Present24
			AND NOT Part_Present25 AND NOT Part_Present26 AND NOT Part_Present27
			AND NOT Part_Present28 AND NOT Part_Present29 AND NOT Part_Present30
			AND NOT Part_Present31 AND NOT Part_Present32 AND NOT Part_Present33
			AND NOT Part_Present34 AND NOT Part_Present35 AND NOT Part_Present36
			AND NOT Part_Present37 AND NOT Part_Present38 AND NOT Part_Present39
			AND NOT Part_Present40;

	(*All Sensors Required Off - Used for sub fixtures where the part has to move from one stage to the next*)
	All_Sensors_Off2:= NOT Part_Present1 AND NOT Part_Present2 AND NOT  Part_Present3
			AND NOT Part_Present4 AND NOT Part_Present5 AND NOT Part_Present6
			AND NOT Part_Present7 AND NOT Part_Present8 AND NOT Part_Present9
			AND NOT Part_Present10 AND NOT Part_Present11 AND NOT Part_Present12
			AND NOT Part_Present13 AND NOT Part_Present14 AND NOT Part_Present15
			AND NOT Part_Present16 AND NOT Part_Present17 AND NOT Part_Present18
			AND NOT Part_Present19 AND NOT Part_Present20 AND NOT Part_Present21
			AND NOT Part_Present22 AND NOT Part_Present23 AND NOT Part_Present24
			AND NOT Part_Present25 AND NOT Part_Present26 AND NOT Part_Present27
			AND NOT Part_Present28 AND NOT Part_Present29 AND NOT Part_Present30
			AND NOT Part_Present31 AND NOT Part_Present32 AND NOT Part_Present33
			AND NOT Part_Present34 AND NOT Part_Present35 AND NOT Part_Present36
			AND NOT Part_Present37 AND NOT Part_Present38 AND NOT Part_Present39
			AND NOT Part_Present40;



(**************************************************************************All Sensors On******************************************************************************)
(**************************************************************************All Sensors On******************************************************************************)
(**************************************************************************All Sensors On******************************************************************************)


	(*Sensors Required for Start Of 1st Robot Load*)
	All_Sensors_On.0:= FALSE OR (Dry_Cycle AND All_Sensors_Off);
	(*Sensors Required for Start of 2nd Robot Load*)
	All_Sensors_On.1:= FALSE OR  (Dry_Cycle AND All_Sensors_Off);

	(*Sensors After Load Complete*)
	All_Sensors_On.2:=(
					((Model_ID=1)
						AND Part_Present1 AND Part_Present2 AND Part_Present3
						AND Part_Present4 AND Part_Present5 AND Part_Present6
						AND Part_Present7 AND Part_Present8 AND Part_Present9
						AND Part_Present10 AND Part_Present11 AND Part_Present12
						AND Part_Present13 AND Part_Present14 AND Part_Present15
						AND Part_Present16 AND Part_Present17 AND Part_Present18
						AND Part_Present19 AND Part_Present20 AND Part_Present21
						AND Part_Present22 AND Part_Present23 AND Part_Present24
						AND Part_Present25 AND Part_Present26 AND Part_Present27
						AND Part_Present28 AND Part_Present29 AND Part_Present30
						AND Part_Present31 AND Part_Present32 AND Part_Present33
						AND Part_Present34 AND Part_Present35 AND Part_Present36
						AND Part_Present37 AND Part_Present38 AND Part_Present39
						AND Part_Present40)

					OR ((Model_ID=2)
						AND Part_Present1 AND Part_Present2 AND Part_Present3
						AND Part_Present4 AND Part_Present5 AND Part_Present6
						AND Part_Present7 AND Part_Present8 AND Part_Present9
						AND Part_Present10 AND Part_Present11 AND Part_Present12
						AND Part_Present13 AND Part_Present14 AND Part_Present15
						AND Part_Present16 AND Part_Present17 AND Part_Present18
						AND Part_Present19 AND Part_Present20 AND Part_Present21
						AND Part_Present22 AND Part_Present23 AND Part_Present24
						AND Part_Present25 AND Part_Present26 AND Part_Present27
						AND Part_Present28 AND Part_Present29 AND Part_Present30
						AND Part_Present31 AND Part_Present32 AND Part_Present33
						AND Part_Present34 AND Part_Present35 AND Part_Present36
						AND Part_Present37 AND Part_Present38 AND Part_Present39
						AND Part_Present40)

					OR ((Model_ID=3)
						AND Part_Present1 AND Part_Present2 AND Part_Present3
						AND Part_Present4 AND Part_Present5 AND Part_Present6
						AND Part_Present7 AND Part_Present8 AND Part_Present9
						AND Part_Present10 AND Part_Present11 AND Part_Present12
						AND Part_Present13 AND Part_Present14 AND Part_Present15
						AND Part_Present16 AND Part_Present17 AND Part_Present18
						AND Part_Present19 AND Part_Present20 AND Part_Present21
						AND Part_Present22 AND Part_Present23 AND Part_Present24
						AND Part_Present25 AND Part_Present26 AND Part_Present27
						AND Part_Present28 AND Part_Present29 AND Part_Present30
						AND Part_Present31 AND Part_Present32 AND Part_Present33
						AND Part_Present34 AND Part_Present35 AND Part_Present36
						AND Part_Present37 AND Part_Present38 AND Part_Present39
						AND Part_Present40)

					OR ((Model_ID=4)
						AND Part_Present1 AND Part_Present2 AND Part_Present3
						AND Part_Present4 AND Part_Present5 AND Part_Present6
						AND Part_Present7 AND Part_Present8 AND Part_Present9
						AND Part_Present10 AND Part_Present11 AND Part_Present12
						AND Part_Present13 AND Part_Present14 AND Part_Present15
						AND Part_Present16 AND Part_Present17 AND Part_Present18
						AND Part_Present19 AND Part_Present20 AND Part_Present21
						AND Part_Present22 AND Part_Present23 AND Part_Present24
						AND Part_Present25 AND Part_Present26 AND Part_Present27
						AND Part_Present28 AND Part_Present29 AND Part_Present30
						AND Part_Present31 AND Part_Present32 AND Part_Present33
						AND Part_Present34 AND Part_Present35 AND Part_Present36
						AND Part_Present37 AND Part_Present38 AND Part_Present39
						AND Part_Present40)
					) OR (All_Sensors_Off AND Dry_Cycle);


	(*Sensors Require for Start Of Welding*)
	All_Sensors_On.3:=(
					((Model_ID=1)
						AND Part_Present1 AND Part_Present2 AND Part_Present3
						AND Part_Present4 AND Part_Present5 AND Part_Present6
						AND Part_Present7 AND Part_Present8 AND Part_Present9
						AND Part_Present10 AND Part_Present11 AND Part_Present12
						AND Part_Present13 AND Part_Present14 AND Part_Present15
						AND Part_Present16 AND Part_Present17 AND Part_Present18
						AND Part_Present19 AND Part_Present20 AND Part_Present21
						AND Part_Present22 AND Part_Present23 AND Part_Present24
						AND Part_Present25 AND Part_Present26 AND Part_Present27
						AND Part_Present28 AND Part_Present29 AND Part_Present30
						AND Part_Present31 AND Part_Present32 AND Part_Present33
						AND Part_Present34 AND Part_Present35 AND Part_Present36
						AND Part_Present37 AND Part_Present38 AND Part_Present39
						AND Part_Present40)

					OR ((Model_ID=2)
						AND Part_Present1 AND Part_Present2 AND Part_Present3
						AND Part_Present4 AND Part_Present5 AND Part_Present6
						AND Part_Present7 AND Part_Present8 AND Part_Present9
						AND Part_Present10 AND Part_Present11 AND Part_Present12
						AND Part_Present13 AND Part_Present14 AND Part_Present15
						AND Part_Present16 AND Part_Present17 AND Part_Present18
						AND Part_Present19 AND Part_Present20 AND Part_Present21
						AND Part_Present22 AND Part_Present23 AND Part_Present24
						AND Part_Present25 AND Part_Present26 AND Part_Present27
						AND Part_Present28 AND Part_Present29 AND Part_Present30
						AND Part_Present31 AND Part_Present32 AND Part_Present33
						AND Part_Present34 AND Part_Present35 AND Part_Present36
						AND Part_Present37 AND Part_Present38 AND Part_Present39
						AND Part_Present40)

					OR ((Model_ID=3)
						AND Part_Present1 AND Part_Present2 AND Part_Present3
						AND Part_Present4 AND Part_Present5 AND Part_Present6
						AND Part_Present7 AND Part_Present8 AND Part_Present9
						AND Part_Present10 AND Part_Present11 AND Part_Present12
						AND Part_Present13 AND Part_Present14 AND Part_Present15
						AND Part_Present16 AND Part_Present17 AND Part_Present18
						AND Part_Present19 AND Part_Present20 AND Part_Present21
						AND Part_Present22 AND Part_Present23 AND Part_Present24
						AND Part_Present25 AND Part_Present26 AND Part_Present27
						AND Part_Present28 AND Part_Present29 AND Part_Present30
						AND Part_Present31 AND Part_Present32 AND Part_Present33
						AND Part_Present34 AND Part_Present35 AND Part_Present36
						AND Part_Present37 AND Part_Present38 AND Part_Present39
						AND Part_Present40)

					OR ((Model_ID=4)
						AND Part_Present1 AND Part_Present2 AND Part_Present3
						AND Part_Present4 AND Part_Present5 AND Part_Present6
						AND Part_Present7 AND Part_Present8 AND Part_Present9
						AND Part_Present10 AND Part_Present11 AND Part_Present12
						AND Part_Present13 AND Part_Present14 AND Part_Present15
						AND Part_Present16 AND Part_Present17 AND Part_Present18
						AND Part_Present19 AND Part_Present20 AND Part_Present21
						AND Part_Present22 AND Part_Present23 AND Part_Present24
						AND Part_Present25 AND Part_Present26 AND Part_Present27
						AND Part_Present28 AND Part_Present29 AND Part_Present30
						AND Part_Present31 AND Part_Present32 AND Part_Present33
						AND Part_Present34 AND Part_Present35 AND Part_Present36
						AND Part_Present37 AND Part_Present38 AND Part_Present39
						AND Part_Present40)
					) OR (All_Sensors_Off AND Dry_Cycle);


	(*Sensors Required After Repo_Reqs.0*)
	All_Sensors_On.4:= (FALSE) OR (Dry_Cycle AND All_Sensors_Off);
	(*Sensors Required After Repo_Reqs.1*)
	All_Sensors_On.5:= (FALSE) OR (Dry_Cycle AND All_Sensors_Off);
	(*Sensors Required After Repo_Reqs.2*)
	All_Sensors_On.6:= (FALSE) OR (Dry_Cycle AND All_Sensors_Off);
	(*Sensors Required After Repo_Reqs.3*)
	All_Sensors_On.7:= (FALSE) OR (Dry_Cycle AND All_Sensors_Off);


	(*Sensors Required for Start Of Unload1*)
	All_Sensors_On.8:=(
					((Model_ID=1)
						AND Part_Present1 AND Part_Present2 AND Part_Present3
						AND Part_Present4 AND Part_Present5 AND Part_Present6
						AND Part_Present7 AND Part_Present8 AND Part_Present9
						AND Part_Present10 AND Part_Present11 AND Part_Present12
						AND Part_Present13 AND Part_Present14 AND Part_Present15
						AND Part_Present16 AND Part_Present17 AND Part_Present18
						AND Part_Present19 AND Part_Present20 AND Part_Present21
						AND Part_Present22 AND Part_Present23 AND Part_Present24
						AND Part_Present25 AND Part_Present26 AND Part_Present27
						AND Part_Present28 AND Part_Present29 AND Part_Present30
						AND Part_Present31 AND Part_Present32 AND Part_Present33
						AND Part_Present34 AND Part_Present35 AND Part_Present36
						AND Part_Present37 AND Part_Present38 AND Part_Present39
						AND Part_Present40)

					OR ((Model_ID=2)
						AND Part_Present1 AND Part_Present2 AND Part_Present3
						AND Part_Present4 AND Part_Present5 AND Part_Present6
						AND Part_Present7 AND Part_Present8 AND Part_Present9
						AND Part_Present10 AND Part_Present11 AND Part_Present12
						AND Part_Present13 AND Part_Present14 AND Part_Present15
						AND Part_Present16 AND Part_Present17 AND Part_Present18
						AND Part_Present19 AND Part_Present20 AND Part_Present21
						AND Part_Present22 AND Part_Present23 AND Part_Present24
						AND Part_Present25 AND Part_Present26 AND Part_Present27
						AND Part_Present28 AND Part_Present29 AND Part_Present30
						AND Part_Present31 AND Part_Present32 AND Part_Present33
						AND Part_Present34 AND Part_Present35 AND Part_Present36
						AND Part_Present37 AND Part_Present38 AND Part_Present39
						AND Part_Present40)

					OR ((Model_ID=3)
						AND Part_Present1 AND Part_Present2 AND Part_Present3
						AND Part_Present4 AND Part_Present5 AND Part_Present6
						AND Part_Present7 AND Part_Present8 AND Part_Present9
						AND Part_Present10 AND Part_Present11 AND Part_Present12
						AND Part_Present13 AND Part_Present14 AND Part_Present15
						AND Part_Present16 AND Part_Present17 AND Part_Present18
						AND Part_Present19 AND Part_Present20 AND Part_Present21
						AND Part_Present22 AND Part_Present23 AND Part_Present24
						AND Part_Present25 AND Part_Present26 AND Part_Present27
						AND Part_Present28 AND Part_Present29 AND Part_Present30
						AND Part_Present31 AND Part_Present32 AND Part_Present33
						AND Part_Present34 AND Part_Present35 AND Part_Present36
						AND Part_Present37 AND Part_Present38 AND Part_Present39
						AND Part_Present40)

					OR ((Model_ID=4)
						AND Part_Present1 AND Part_Present2 AND Part_Present3
						AND Part_Present4 AND Part_Present5 AND Part_Present6
						AND Part_Present7 AND Part_Present8 AND Part_Present9
						AND Part_Present10 AND Part_Present11 AND Part_Present12
						AND Part_Present13 AND Part_Present14 AND Part_Present15
						AND Part_Present16 AND Part_Present17 AND Part_Present18
						AND Part_Present19 AND Part_Present20 AND Part_Present21
						AND Part_Present22 AND Part_Present23 AND Part_Present24
						AND Part_Present25 AND Part_Present26 AND Part_Present27
						AND Part_Present28 AND Part_Present29 AND Part_Present30
						AND Part_Present31 AND Part_Present32 AND Part_Present33
						AND Part_Present34 AND Part_Present35 AND Part_Present36
						AND Part_Present37 AND Part_Present38 AND Part_Present39
						AND Part_Present40)
					) OR (All_Sensors_Off AND Dry_Cycle);

	(*Sensors Required for Start Of Unload2*)
	All_Sensors_On.9:=(
					((Model_ID=1)
						AND Part_Present1 AND Part_Present2 AND Part_Present3
						AND Part_Present4 AND Part_Present5 AND Part_Present6
						AND Part_Present7 AND Part_Present8 AND Part_Present9
						AND Part_Present10 AND Part_Present11 AND Part_Present12
						AND Part_Present13 AND Part_Present14 AND Part_Present15
						AND Part_Present16 AND Part_Present17 AND Part_Present18
						AND Part_Present19 AND Part_Present20 AND Part_Present21
						AND Part_Present22 AND Part_Present23 AND Part_Present24
						AND Part_Present25 AND Part_Present26 AND Part_Present27
						AND Part_Present28 AND Part_Present29 AND Part_Present30
						AND Part_Present31 AND Part_Present32 AND Part_Present33
						AND Part_Present34 AND Part_Present35 AND Part_Present36
						AND Part_Present37 AND Part_Present38 AND Part_Present39
						AND Part_Present40)

					OR ((Model_ID=2)
						AND Part_Present1 AND Part_Present2 AND Part_Present3
						AND Part_Present4 AND Part_Present5 AND Part_Present6
						AND Part_Present7 AND Part_Present8 AND Part_Present9
						AND Part_Present10 AND Part_Present11 AND Part_Present12
						AND Part_Present13 AND Part_Present14 AND Part_Present15
						AND Part_Present16 AND Part_Present17 AND Part_Present18
						AND Part_Present19 AND Part_Present20 AND Part_Present21
						AND Part_Present22 AND Part_Present23 AND Part_Present24
						AND Part_Present25 AND Part_Present26 AND Part_Present27
						AND Part_Present28 AND Part_Present29 AND Part_Present30
						AND Part_Present31 AND Part_Present32 AND Part_Present33
						AND Part_Present34 AND Part_Present35 AND Part_Present36
						AND Part_Present37 AND Part_Present38 AND Part_Present39
						AND Part_Present40)

					OR ((Model_ID=3)
						AND Part_Present1 AND Part_Present2 AND Part_Present3
						AND Part_Present4 AND Part_Present5 AND Part_Present6
						AND Part_Present7 AND Part_Present8 AND Part_Present9
						AND Part_Present10 AND Part_Present11 AND Part_Present12
						AND Part_Present13 AND Part_Present14 AND Part_Present15
						AND Part_Present16 AND Part_Present17 AND Part_Present18
						AND Part_Present19 AND Part_Present20 AND Part_Present21
						AND Part_Present22 AND Part_Present23 AND Part_Present24
						AND Part_Present25 AND Part_Present26 AND Part_Present27
						AND Part_Present28 AND Part_Present29 AND Part_Present30
						AND Part_Present31 AND Part_Present32 AND Part_Present33
						AND Part_Present34 AND Part_Present35 AND Part_Present36
						AND Part_Present37 AND Part_Present38 AND Part_Present39
						AND Part_Present40)

					OR ((Model_ID=4)
						AND Part_Present1 AND Part_Present2 AND Part_Present3
						AND Part_Present4 AND Part_Present5 AND Part_Present6
						AND Part_Present7 AND Part_Present8 AND Part_Present9
						AND Part_Present10 AND Part_Present11 AND Part_Present12
						AND Part_Present13 AND Part_Present14 AND Part_Present15
						AND Part_Present16 AND Part_Present17 AND Part_Present18
						AND Part_Present19 AND Part_Present20 AND Part_Present21
						AND Part_Present22 AND Part_Present23 AND Part_Present24
						AND Part_Present25 AND Part_Present26 AND Part_Present27
						AND Part_Present28 AND Part_Present29 AND Part_Present30
						AND Part_Present31 AND Part_Present32 AND Part_Present33
						AND Part_Present34 AND Part_Present35 AND Part_Present36
						AND Part_Present37 AND Part_Present38 AND Part_Present39
						AND Part_Present40)
					) OR (All_Sensors_Off AND Dry_Cycle);


























(*end*)
END_ACTION

ACTION Cylinders:

(* -----------------------------------------------------------------------------------*)
(*Below are Examples only, each will have to be customized for your application
	Notes:
	- Use SODGxx-SSCC61x-xxxxxxx_Fix IO and Seq.xlsx document to capture Clamp / Cylinder I/O Layout
	- CLFaults1 thru 4 can be used to group cylinder type faults (All Clamps on CLFaults1, all Pins on CLFaults2)
		OR
	- CLFaults 1 thru 4 can be used to group cylinder UI screens 
		(All items on Cylinder_1.content screen are on CLFaults1, all items on Cylinder_2.content screen are on CLFaults2 as example)
*)
(* -----------------------------------------------------------------------------------*)



(*Clamps*)(*Clamps*)(*Clamps*)
(*Clamps*)(*Clamps*)(*Clamps*)
(*Clamps*)(*Clamps*)(*Clamps*)

		(*Clamp1*)
		Clamp1FB(
			Retracted_Sensor:= N02.I.0 ,
			Advanced_Sensor:= N02.I.1 ,
			Retract_Solenoid:= N100.Q.1,
			Advance_Solenoid:= N100.Q.0 ,
			Ret_Delay:= T#0.1S,
			Adv_Delay:= T#0.1S,
			Fault_Delay:= T#3.0S,
			Disable_Fault:= FALSE,
			In_Retracted_Position=> Clamp1RETD,
			In_Advanced_Position=> Clamp1ADVD,
			Faulted=> CLFaults1.1 );

		(*Clamp2*)
		Clamp2FB(
			Retracted_Sensor:= N02.I.2 ,
			Advanced_Sensor:= N02.I.3 ,
			Retract_Solenoid:= N100.Q.1 ,
			Advance_Solenoid:= N100.Q.0 ,
			Ret_Delay:= T#0.1S,
			Adv_Delay:= T#0.1S,
			Fault_Delay:= T#3.0S,
			Disable_Fault:= FALSE,
			In_Retracted_Position=> Clamp2RETD,
			In_Advanced_Position=> Clamp2ADVD,
			Faulted=> CLFaults1.2 );

		(*Clamp3*)
		Clamp3FB(
			Retracted_Sensor:= N02.I.4,
			Advanced_Sensor:= N02.I.5,
			Retract_Solenoid:= N100.Q.1,
			Advance_Solenoid:= N100.Q.0,
			Ret_Delay:= T#0.1S,
			Adv_Delay:= T#0.1S,
			Fault_Delay:= T#3.0S,
			Disable_Fault:= FALSE,
			In_Retracted_Position=> Clamp3RETD,
			In_Advanced_Position=> Clamp3ADVD,
			Faulted=> CLFaults1.3 );

		(*Clamp4*)
		Clamp4FB(
			Retracted_Sensor:= N02.I.6,
			Advanced_Sensor:= N02.I.7,
			Retract_Solenoid:= N100.Q.1,
			Advance_Solenoid:= N100.Q.0,
			Ret_Delay:= T#0.1S,
			Adv_Delay:= T#0.1S,
			Fault_Delay:= T#3.0S,
			Disable_Fault:= FALSE,
			In_Retracted_Position=> Clamp4RETD,
			In_Advanced_Position=> Clamp4ADVD,
			Faulted=> CLFaults1.4 );

		(*Clamp5*)
		Clamp5FB(
			Retracted_Sensor:= N03.I.0,
			Advanced_Sensor:= N03.I.1,
			Retract_Solenoid:= N100.Q.1,
			Advance_Solenoid:= N100.Q.0,
			Ret_Delay:= T#0.1S,
			Adv_Delay:= T#0.1S,
			Fault_Delay:= T#3.0S,
			Disable_Fault:= FALSE,
			In_Retracted_Position=> Clamp5RETD,
			In_Advanced_Position=> Clamp5ADVD,
			Faulted=> CLFaults1.5 );

		(*Clamp6*)
		Clamp6FB(
			Retracted_Sensor:= N03.I.2,
			Advanced_Sensor:= N03.I.3,
			Retract_Solenoid:= N100.Q.1,
			Advance_Solenoid:= N100.Q.0,
			Ret_Delay:= T#0.1S,
			Adv_Delay:= T#0.1S,
			Fault_Delay:= T#3.0S,
			Disable_Fault:= FALSE,
			In_Retracted_Position=> Clamp6RETD,
			In_Advanced_Position=> Clamp6ADVD,
			Faulted=> CLFaults1.6 );

		(*Clamp7*)
		Clamp7FB(
			Retracted_Sensor:= N03.I.4,
			Advanced_Sensor:= N03.I.5,
			Retract_Solenoid:= N100.Q.1,
			Advance_Solenoid:= N100.Q.0,
			Ret_Delay:= T#0.1S,
			Adv_Delay:= T#0.1S,
			Fault_Delay:= T#3.0S,
			Disable_Fault:= FALSE,
			In_Retracted_Position=> Clamp7RETD,
			In_Advanced_Position=> Clamp7ADVD,
			Faulted=> CLFaults1.7 );

		(*Clamp8*)
		Clamp8FB(
			Retracted_Sensor:= N03.I.6,
			Advanced_Sensor:= N03.I.7,
			Retract_Solenoid:= N100.Q.1,
			Advance_Solenoid:= N100.Q.0,
			Ret_Delay:= T#0.1S,
			Adv_Delay:= T#0.1S,
			Fault_Delay:= T#3.0S,
			Disable_Fault:= FALSE,
			In_Retracted_Position=> Clamp8RETD,
			In_Advanced_Position=> Clamp8ADVD,
			Faulted=> CLFaults1.8 );

		(*Clamp9*)
		Clamp9FB(
			Retracted_Sensor:= N04.I.0,
			Advanced_Sensor:= N04.I.1,
			Retract_Solenoid:= N100.Q.3,
			Advance_Solenoid:= N100.Q.2,
			Ret_Delay:= T#0.1S,
			Adv_Delay:= T#0.1S,
			Fault_Delay:= T#3.0S,
			Disable_Fault:= FALSE,
			In_Retracted_Position=> Clamp9RETD,
			In_Advanced_Position=> Clamp9ADVD,
			Faulted=> CLFaults1.9 );

		(*Clamp10*)
		Clamp10FB(
			Retracted_Sensor:= N04.I.2,
			Advanced_Sensor:= N04.I.3,
			Retract_Solenoid:= N100.Q.3,
			Advance_Solenoid:= N100.Q.2,
			Ret_Delay:= T#0.1S,
			Adv_Delay:= T#0.1S,
			Fault_Delay:= T#3.0S,
			Disable_Fault:= FALSE,
			In_Retracted_Position=> Clamp10RETD,
			In_Advanced_Position=> Clamp10ADVD,
			Faulted=> CLFaults1.10 );

		(*Clamp11*)
		Clamp11FB(
			Retracted_Sensor:= N04.I.4,
			Advanced_Sensor:= N04.I.5,
			Retract_Solenoid:= N100.Q.3,
			Advance_Solenoid:= N100.Q.2,
			Ret_Delay:= T#0.1S,
			Adv_Delay:= T#0.1S,
			Fault_Delay:= T#3.0S,
			Disable_Fault:= FALSE,
			In_Retracted_Position=> Clamp11RETD,
			In_Advanced_Position=> Clamp11ADVD,
			Faulted=> CLFaults1.11 );

		(*Clamp12*)
		Clamp12FB(
			Retracted_Sensor:= N04.I.6,
			Advanced_Sensor:= N04.I.7,
			Retract_Solenoid:= N100.Q.3,
			Advance_Solenoid:= N100.Q.2,
			Ret_Delay:= T#0.1S,
			Adv_Delay:= T#0.1S,
			Fault_Delay:= T#3.0S,
			Disable_Fault:= FALSE,
			In_Retracted_Position=> Clamp12RETD,
			In_Advanced_Position=> Clamp12ADVD,
			Faulted=> CLFaults1.12 );

		(*Clamp13*)
		Clamp13FB(
			Retracted_Sensor:= N05.I.0,
			Advanced_Sensor:= N05.I.1,
			Retract_Solenoid:= N100.Q.5,
			Advance_Solenoid:= N100.Q.4,
			Ret_Delay:= T#0.1S,
			Adv_Delay:= T#0.1S,
			Fault_Delay:= T#3.0S,
			Disable_Fault:= FALSE,
			In_Retracted_Position=> Clamp13RETD,
			In_Advanced_Position=> Clamp13ADVD,
			Faulted=> CLFaults1.13 );

		(*Clamp14*)
		Clamp14FB(
			Retracted_Sensor:= N05.I.2,
			Advanced_Sensor:= N05.I.3,
			Retract_Solenoid:= N100.Q.5,
			Advance_Solenoid:= N100.Q.4,
			Ret_Delay:= T#0.1S,
			Adv_Delay:= T#0.1S,
			Fault_Delay:= T#3.0S,
			Disable_Fault:= FALSE,
			In_Retracted_Position=> Clamp14RETD,
			In_Advanced_Position=> Clamp14ADVD,
			Faulted=> CLFaults1.14 );

		(*Clamp15*)
		Clamp15FB(
			Retracted_Sensor:= N05.I.4,
			Advanced_Sensor:= N05.I.5,
			Retract_Solenoid:= N100.Q.5,
			Advance_Solenoid:= N100.Q.4,
			Ret_Delay:= T#0.1S,
			Adv_Delay:= T#0.1S,
			Fault_Delay:= T#3.0S,
			Disable_Fault:= FALSE,
			In_Retracted_Position=> Clamp15RETD,
			In_Advanced_Position=> Clamp15ADVD,
			Faulted=> CLFaults1.15 );

		(*Clamp16*)
		Clamp16FB(
			Retracted_Sensor:= N05.I.6,
			Advanced_Sensor:= N05.I.7,
			Retract_Solenoid:= N100.Q.5,
			Advance_Solenoid:= N100.Q.4,
			Ret_Delay:= T#0.1S,
			Adv_Delay:= T#0.1S,
			Fault_Delay:= T#3.0S,
			Disable_Fault:= FALSE,
			In_Retracted_Position=> Clamp16RETD,
			In_Advanced_Position=> Clamp16ADVD,
			Faulted=> CLFaults1.16 );

		(*Clamp17*)
		Clamp17FB(
			Retracted_Sensor:= N06.I.0,
			Advanced_Sensor:= N06.I.1,
			Retract_Solenoid:= N100.Q.7,
			Advance_Solenoid:= N100.Q.6,
			Ret_Delay:= T#0.1S,
			Adv_Delay:= T#0.1S,
			Fault_Delay:= T#3.0S,
			Disable_Fault:= FALSE,
			In_Retracted_Position=> Clamp17RETD,
			In_Advanced_Position=> Clamp17ADVD,
			Faulted=> CLFaults1.17 );

		(*Clamp18*)
		Clamp18FB(
			Retracted_Sensor:= N06.I.2,
			Advanced_Sensor:= N06.I.3,
			Retract_Solenoid:= N100.Q.7,
			Advance_Solenoid:= N100.Q.6,
			Ret_Delay:= T#0.1S,
			Adv_Delay:= T#0.1S,
			Fault_Delay:= T#3.0S,
			Disable_Fault:= FALSE,
			In_Retracted_Position=> Clamp18RETD,
			In_Advanced_Position=> Clamp18ADVD,
			Faulted=> CLFaults1.18 );

		(*Clamp19*)
		Clamp19FB(
			Retracted_Sensor:= N06.I.4,
			Advanced_Sensor:= N06.I.5,
			Retract_Solenoid:= N100.Q.7,
			Advance_Solenoid:= N100.Q.6,
			Ret_Delay:= T#0.1S,
			Adv_Delay:= T#0.1S,
			Fault_Delay:= T#3.0S,
			Disable_Fault:= FALSE,
			In_Retracted_Position=> Clamp19RETD,
			In_Advanced_Position=> Clamp19ADVD,
			Faulted=> CLFaults1.19 );

		(*Clamp20*)
		Clamp20FB(
			Retracted_Sensor:= N06.I.6,
			Advanced_Sensor:= N06.I.7,
			Retract_Solenoid:= N100.Q.7,
			Advance_Solenoid:= N100.Q.6,
			Ret_Delay:= T#0.1S,
			Adv_Delay:= T#0.1S,
			Fault_Delay:= T#3.0S,
			Disable_Fault:= FALSE,
			In_Retracted_Position=> Clamp20RETD,
			In_Advanced_Position=> Clamp20ADVD,
			Faulted=> CLFaults1.20 );

		(*Clamp21*)
		Clamp21FB(
			Retracted_Sensor:= N07.I.0,
			Advanced_Sensor:= N07.I.1,
			Retract_Solenoid:= N100.Q.9,
			Advance_Solenoid:= N100.Q.8,
			Ret_Delay:= T#0.1S,
			Adv_Delay:= T#0.1S,
			Fault_Delay:= T#3.0S,
			Disable_Fault:= FALSE,
			In_Retracted_Position=> Clamp21RETD,
			In_Advanced_Position=> Clamp21ADVD,
			Faulted=> CLFaults1.21 );

		(*Clamp22*)
		Clamp22FB(
			Retracted_Sensor:= N07.I.2,
			Advanced_Sensor:= N07.I.3,
			Retract_Solenoid:= N100.Q.9,
			Advance_Solenoid:= N100.Q.8,
			Ret_Delay:= T#0.1S,
			Adv_Delay:= T#0.1S,
			Fault_Delay:= T#3.0S,
			Disable_Fault:= FALSE,
			In_Retracted_Position=> Clamp22RETD,
			In_Advanced_Position=> Clamp22ADVD,
			Faulted=> CLFaults1.22 );

		(*Clamp23*)
		Clamp23FB(
			Retracted_Sensor:= N07.I.4,
			Advanced_Sensor:= N07.I.5,
			Retract_Solenoid:= N100.Q.9,
			Advance_Solenoid:= N100.Q.8,
			Ret_Delay:= T#0.1S,
			Adv_Delay:= T#0.1S,
			Fault_Delay:= T#3.0S,
			Disable_Fault:= FALSE,
			In_Retracted_Position=> Clamp23RETD,
			In_Advanced_Position=> Clamp23ADVD,
			Faulted=> CLFaults1.23 );

		(*Clamp24*)
		Clamp24FB(
			Retracted_Sensor:= N07.I.6,
			Advanced_Sensor:= N07.I.7,
			Retract_Solenoid:= N100.Q.9,
			Advance_Solenoid:= N100.Q.8,
			Ret_Delay:= T#0.1S,
			Adv_Delay:= T#0.1S,
			Fault_Delay:= T#3.0S,
			Disable_Fault:= FALSE,
			In_Retracted_Position=> Clamp24RETD,
			In_Advanced_Position=> Clamp24ADVD,
			Faulted=> CLFaults1.24 );


(*Pins*)(*Pins*)(*Pins*)
(*Pins*)(*Pins*)(*Pins*)
(*Pins*)(*Pins*)(*Pins*)

		(*Pin1*)
		Pin1FB(
			Retracted_Sensor:= N03.I.0,
			Advanced_Sensor:= N03.I.1,
			Retract_Solenoid:= N101.Q.1,
			Advance_Solenoid:= N101.Q.0,
			Ret_Delay:= T#0.1S,
			Adv_Delay:= T#0.1S,
			Fault_Delay:= T#3.0S,
			Disable_Fault:= FALSE,
			In_Retracted_Position=> Pin1RETD,
			In_Advanced_Position=> Pin1ADVD,
			Faulted=> CLFaults2.1 );

		(*Pin2*)
		Pin2FB(
			Retracted_Sensor:= N03.I.2,
			Advanced_Sensor:= N03.I.3,
			Retract_Solenoid:= N101.Q.1,
			Advance_Solenoid:= N101.Q.0,
			Ret_Delay:= T#0.1S,
			Adv_Delay:= T#0.1S,
			Fault_Delay:= T#3.0S,
			Disable_Fault:= FALSE,
			In_Retracted_Position=> Pin2RETD,
			In_Advanced_Position=> Pin2ADVD,
			Faulted=> CLFaults2.2 );

		(*Pin3*)
		Pin3FB(
			Retracted_Sensor:= N03.I.4,
			Advanced_Sensor:= N03.I.5,
			Retract_Solenoid:= N101.Q.1,
			Advance_Solenoid:= N101.Q.0,
			Ret_Delay:= T#0.1S,
			Adv_Delay:= T#0.1S,
			Fault_Delay:= T#3.0S,
			Disable_Fault:= FALSE,
			In_Retracted_Position=> Pin3RETD,
			In_Advanced_Position=> Pin3ADVD,
			Faulted=> CLFaults2.3 );

		(*Pin4*)
		Pin4FB(
			Retracted_Sensor:= N03.I.6,
			Advanced_Sensor:= N10.I.7,
			Retract_Solenoid:= N101.Q.1,
			Advance_Solenoid:= N101.Q.0,
			Ret_Delay:= T#0.1S,
			Adv_Delay:= T#0.1S,
			Fault_Delay:= T#3.0S,
			Disable_Fault:= FALSE,
			In_Retracted_Position=> Pin4RETD,
			In_Advanced_Position=> Pin4ADVD,
			Faulted=> CLFaults2.4 );

		(*Pin5*)
		Pin5FB(
			Retracted_Sensor:= N04.I.0,
			Advanced_Sensor:= N04.I.1,
			Retract_Solenoid:= N101.Q.1,
			Advance_Solenoid:= N101.Q.0,
			Ret_Delay:= T#0.1S,
			Adv_Delay:= T#0.1S,
			Fault_Delay:= T#3.0S,
			Disable_Fault:= FALSE,
			In_Retracted_Position=> Pin5RETD,
			In_Advanced_Position=> Pin5ADVD,
			Faulted=> CLFaults2.5 );

		(*Pin6*)
		Pin6FB(
			Retracted_Sensor:= N04.I.2,
			Advanced_Sensor:= N04.I.3,
			Retract_Solenoid:= N101.Q.1,
			Advance_Solenoid:= N101.Q.0,
			Ret_Delay:= T#0.1S,
			Adv_Delay:= T#0.1S,
			Fault_Delay:= T#3.0S,
			Disable_Fault:= FALSE,
			In_Retracted_Position=> Pin6RETD,
			In_Advanced_Position=> Pin6ADVD,
			Faulted=> CLFaults2.6 );

		(*Pin7*)
		Pin7FB(
			Retracted_Sensor:= N04.I.4,
			Advanced_Sensor:= N04.I.5,
			Retract_Solenoid:= N101.Q.1,
			Advance_Solenoid:= N101.Q.0,
			Ret_Delay:= T#0.1S,
			Adv_Delay:= T#0.1S,
			Fault_Delay:= T#3.0S,
			Disable_Fault:= FALSE,
			In_Retracted_Position=> Pin7RETD,
			In_Advanced_Position=> Pin7ADVD,
			Faulted=> CLFaults2.7 );

		(*Pin8*)
		Pin8FB(
			Retracted_Sensor:= N04.I.6,
			Advanced_Sensor:= N04.I.7,
			Retract_Solenoid:= N101.Q.1,
			Advance_Solenoid:= N101.Q.0,
			Ret_Delay:= T#0.1S,
			Adv_Delay:= T#0.1S,
			Fault_Delay:= T#3.0S,
			Disable_Fault:= FALSE,
			In_Retracted_Position=> Pin8RETD,
			In_Advanced_Position=> Pin8ADVD,
			Faulted=> CLFaults2.8 );

		(*Pin9*)
		Pin9FB(
			Retracted_Sensor:= N05.I.0,
			Advanced_Sensor:= N05.I.1,
			Retract_Solenoid:= N101.Q.3,
			Advance_Solenoid:= N101.Q.2,
			Ret_Delay:= T#0.1S,
			Adv_Delay:= T#0.1S,
			Fault_Delay:= T#3.0S,
			Disable_Fault:= FALSE,
			In_Retracted_Position=> Pin9RETD,
			In_Advanced_Position=> Pin9ADVD,
			Faulted=> CLFaults2.9 );

		(*Pin10*)
		Pin10FB(
			Retracted_Sensor:= N05.I.2,
			Advanced_Sensor:= N05.I.3,
			Retract_Solenoid:= N101.Q.3,
			Advance_Solenoid:= N101.Q.2,
			Ret_Delay:= T#0.1S,
			Adv_Delay:= T#0.1S,
			Fault_Delay:= T#3.0S,
			Disable_Fault:= FALSE,
			In_Retracted_Position=> Pin10RETD,
			In_Advanced_Position=> Pin10ADVD,
			Faulted=> CLFaults2.10 );

		(*Pin11*)
		Pin11FB(
			Retracted_Sensor:= N05.I.4,
			Advanced_Sensor:= N05.I.5,
			Retract_Solenoid:= N101.Q.3,
			Advance_Solenoid:= N101.Q.2,
			Ret_Delay:= T#0.1S,
			Adv_Delay:= T#0.1S,
			Fault_Delay:= T#3.0S,
			Disable_Fault:= FALSE,
			In_Retracted_Position=> Pin11RETD,
			In_Advanced_Position=> Pin11ADVD,
			Faulted=> CLFaults2.11 );

		(*Pin12*)
		Pin12FB(
			Retracted_Sensor:= N05.I.6,
			Advanced_Sensor:= N05.I.7,
			Retract_Solenoid:= N101.Q.3,
			Advance_Solenoid:= N101.Q.2,
			Ret_Delay:= T#0.1S,
			Adv_Delay:= T#0.1S,
			Fault_Delay:= T#3.0S,
			Disable_Fault:= FALSE,
			In_Retracted_Position=> Pin12RETD,
			In_Advanced_Position=> Pin12ADVD,
			Faulted=> CLFaults2.12 );


(*Slides*)(*Slides*)(*Slides*)
(*Slides*)(*Slides*)(*Slides*)
(*Slides*)(*Slides*)(*Slides*)

		(*Slide1*)
		Slide1FB(
			Retracted_Sensor:= N07.I.0,
			Advanced_Sensor:= N07.I.1,
			Retract_Solenoid:= N100.Q.11,
			Advance_Solenoid:= N100.Q.10,
			Adv_Delay:= T#0.2S,
			Ret_Delay:= T#0.2S,
			Fault_Delay:= T#4.0S,
			Disable_Fault:= FALSE,
			In_Retracted_Position=> Slide1RETD,
			In_Advanced_Position=> Slide1ADVD,
			Faulted=> CLFaults3.1 );

		(*Slide2*)
		Slide2FB(
			Retracted_Sensor:= N07.I.2,
			Advanced_Sensor:= N07.I.3,
			Retract_Solenoid:= N100.Q.11,
			Advance_Solenoid:= N100.Q.10,
			Adv_Delay:= T#0.2S,
			Ret_Delay:= T#0.2S,
			Fault_Delay:= T#4.0S,
			Disable_Fault:= FALSE,
			In_Retracted_Position=> Slide2RETD,
			In_Advanced_Position=> Slide2ADVD,
			Faulted=> CLFaults3.2 );

		(*Slide3*)
		Slide3FB(
			Retracted_Sensor:= N07.I.4,
			Advanced_Sensor:= N07.I.5,
			Retract_Solenoid:= N101.Q.11,
			Advance_Solenoid:= N101.Q.10,
			Adv_Delay:= T#0.2S,
			Ret_Delay:= T#0.2S,
			Fault_Delay:= T#4.0S,
			Disable_Fault:= FALSE,
			In_Retracted_Position=> Slide3RETD,
			In_Advanced_Position=> Slide3ADVD,
			Faulted=> CLFaults3.3 );

		(*Slide4*)
		Slide4FB(
			Retracted_Sensor:= N07.I.6,
			Advanced_Sensor:= N07.I.7,
			Retract_Solenoid:= N101.Q.11,
			Advance_Solenoid:= N101.Q.10,
			Adv_Delay:= T#0.2S,
			Ret_Delay:= T#0.2S,
			Fault_Delay:= T#4.0S,
			Disable_Fault:= FALSE,
			In_Retracted_Position=> Slide4RETD,
			In_Advanced_Position=> Slide4ADVD,
			Faulted=> CLFaults3.4 );

		(*Slide5*)
		Slide5FB(
			Retracted_Sensor:= N08.I.0,
			Advanced_Sensor:= N08.I.1,
			Retract_Solenoid:= N101.Q.11,
			Advance_Solenoid:= N101.Q.10,
			Adv_Delay:= T#0.2S,
			Ret_Delay:= T#0.2S,
			Fault_Delay:= T#4.0S,
			Disable_Fault:= FALSE,
			In_Retracted_Position=> Slide5RETD,
			In_Advanced_Position=> Slide5ADVD,
			Faulted=> CLFaults3.5 );

		(*Slide6*)
		Slide6FB(
			Retracted_Sensor:= N08.I.0,
			Advanced_Sensor:= N08.I.1,
			Retract_Solenoid:= N101.Q.11,
			Advance_Solenoid:= N101.Q.10,
			Adv_Delay:= T#0.2S,
			Ret_Delay:= T#0.2S,
			Fault_Delay:= T#4.0S,
			Disable_Fault:= FALSE,
			In_Retracted_Position=> Slide6RETD,
			In_Advanced_Position=> Slide6ADVD,
			Faulted=> CLFaults3.6 );


(*Swings*)(*Swings*)(*Swings*)
(*Swings*)(*Swings*)(*Swings*)
(*Swings*)(*Swings*)(*Swings*)

		(*Swing1*)
		Swing1FB(
			Retracted_Sensor:= N09.I.0,
			Advanced_Sensor:= N09.I.1,
			Retract_Solenoid:= N101.Q.1,
			Advance_Solenoid:= N101.Q.0,
			Adv_Delay:= T#0.2S,
			Ret_Delay:= T#0.2S,
			Fault_Delay:= T#3.0S,
			Disable_Fault:= FALSE,
			In_Retracted_Position=> Swing1RETD,
			In_Advanced_Position=> Swing1ADVD,
			Faulted=> CLFaults4.1 );

		(*Swing2*)
		Swing2FB(
			Retracted_Sensor:= N09.I.2,
			Advanced_Sensor:= N09.I.3,
			Retract_Solenoid:= N101.Q.3,
			Advance_Solenoid:= N101.Q.2,
			Adv_Delay:= T#0.2S,
			Ret_Delay:= T#0.2S,
			Fault_Delay:= T#3.0S,
			Disable_Fault:= FALSE,
			In_Retracted_Position=> Swing2RETD,
			In_Advanced_Position=> Swing2ADVD,
			Faulted=> CLFaults4.2 );

		(*Swing3*)
		Swing3FB(
			Retracted_Sensor:= N09.I.4,
			Advanced_Sensor:= N09.I.5,
			Retract_Solenoid:= N101.Q.5,
			Advance_Solenoid:= N101.Q.4,
			Adv_Delay:= T#0.2S,
			Ret_Delay:= T#0.2S,
			Fault_Delay:= T#3.0S,
			Disable_Fault:= FALSE,
			In_Retracted_Position=> Swing3RETD,
			In_Advanced_Position=> Swing3ADVD,
			Faulted=> CLFaults4.3 );

		(*Swing4*)
		Swing4FB(
			Retracted_Sensor:= N09.I.6,
			Advanced_Sensor:= N09.I.7,
			Retract_Solenoid:= N101.Q.7,
			Advance_Solenoid:= N101.Q.6,
			Adv_Delay:= T#0.2S,
			Ret_Delay:= T#0.2S,
			Fault_Delay:= T#3.0S,
			Disable_Fault:= FALSE,
			In_Retracted_Position=> Swing4RETD,
			In_Advanced_Position=> Swing4ADVD,
			Faulted=> CLFaults4.4 );

		(*Swing5*)
		Swing5FB(
			Retracted_Sensor:= N10.I.0,
			Advanced_Sensor:= N10.I.1,
			Retract_Solenoid:= N101.Q.9,
			Advance_Solenoid:= N101.Q.8,
			Adv_Delay:= T#0.2S,
			Ret_Delay:= T#0.2S,
			Fault_Delay:= T#3.0S,
			Disable_Fault:= FALSE,
			In_Retracted_Position=> Swing5RETD,
			In_Advanced_Position=> Swing5ADVD,
			Faulted=> CLFaults4.5 );

		(*Swing6*)
		Swing6FB(
			Retracted_Sensor:= N10.I.2,
			Advanced_Sensor:= N10.I.3,
			Retract_Solenoid:= N101.Q.11,
			Advance_Solenoid:= N101.Q.10,
			Adv_Delay:= T#0.2S,
			Ret_Delay:= T#0.2S,
			Fault_Delay:= T#3.0S,
			Disable_Fault:= FALSE,
			In_Retracted_Position=> Swing6RETD,
			In_Advanced_Position=> Swing6ADVD,
			Faulted=> CLFaults4.6 );


(*Triple*)(*Triple*)(*Triple*)
(*Triple*)(*Triple*)(*Triple*)
(*Triple*)(*Triple*)(*Triple*)

		(*Cyl1, Triple Position*)
		Cyl1FB(
			Retracted_Sensor:= N01.I.0,
			Advanced_Sensor:= N01.I.1,
			Mid_Sensor:= N01.I.2,
			Retract_Solenoid:= N100.Q.1,
			Advance_Solenoid:= N100.Q.0,
			Mid_Solenoid:= N100.Q.2,
			Ret_Delay:= T#0.1S,
			Adv_Delay:= T#0.1S,
			Mid_Delay:= T#0.1S,
			Fault_Delay:= T#3.0S,
			Disable_Fault:= FALSE,
			In_Retracted_Position=> Cyl1RETD,
			In_Advanced_Position=> Cyl1ADVD,
			In_Mid_Position=> Cyl1MID,
			Faulted=> CLFaults4.11 );


(*QA*)(*QA*)(*QA*)
(*QA*)(*QA*)(*QA*)
(*QA*)(*QA*)(*QA*)

		(*QA Check1*)
		QACheck1FB(
			Retracted_Sensor:= N04.I.0,
			Advanced_Sensor:= N04.I.1,
			Retract_Solenoid:= N100.Q.5,
			Advance_Solenoid:= N100.Q.4,
			Ret_Delay:= T#0.1S,
			Adv_Delay:= T#0.1S,
			Fault_Delay:= T#3.0S,
			Disable_Fault:= FALSE,
			In_Retracted_Position=> QACheck1RETD,
			In_Advanced_Position=> QACheck1ADVD,
			Faulted=> CLFaults4.1 );

		(*QA Check2*)
		QACheck2FB(
			Retracted_Sensor:= N04.I.2,
			Advanced_Sensor:= N04.I.3,
			Retract_Solenoid:= N100.Q.5,
			Advance_Solenoid:= N100.Q.4,
			Ret_Delay:= T#0.1S,
			Adv_Delay:= T#0.1S,
			Fault_Delay:= T#3.0S,
			Disable_Fault:= FALSE,
			In_Retracted_Position=> QACheck2RETD,
			In_Advanced_Position=> QACheck2ADVD,
			Faulted=> CLFaults4.2 );


(*end*)
END_ACTION

ACTION Hardware:

(*Pass Node States into Array  in order on Physical Fixture*)

		NodeState:=NodeLayout.State;

(*$$$$$$$$$$$$$$$$$$$$$$$$$$$$$$$$$$$$$$$$$$$$$$$$Gather Status Of Hardware $$$$$$$$$$$$$$$$$$$$$$$$$$$$$$$$$$$$$$$$$$$$$$$$$$$$*)

	(*Discrete I/O Nodes*)
	IF N00.InfoData.State=8
		AND (N01.InfoData.State=8 OR (Discrete_In.Input_Node_Count<2))
		AND (N02.InfoData.State=8 OR (Discrete_In.Input_Node_Count<3))
		AND (N03.InfoData.State=8 OR (Discrete_In.Input_Node_Count<4))
		AND (N04.InfoData.State=8 OR (Discrete_In.Input_Node_Count<5))
		AND (N05.InfoData.State=8 OR (Discrete_In.Input_Node_Count<6))
		AND (N06.InfoData.State=8 OR (Discrete_In.Input_Node_Count<7))
		AND (N07.InfoData.State=8 OR (Discrete_In.Input_Node_Count<8))
		AND (N08.InfoData.State=8 OR (Discrete_In.Input_Node_Count<9))
		AND (N09.InfoData.State=8 OR (Discrete_In.Input_Node_Count<10))
		AND (N10.InfoData.State=8 OR (Discrete_In.Input_Node_Count<11))
		AND (N11.InfoData.State=8 OR (Discrete_In.Input_Node_Count<12))
		AND (N12.InfoData.State=8 OR (Discrete_In.Input_Node_Count<13))
		AND (N13.InfoData.State=8 OR (Discrete_In.Input_Node_Count<14))
		AND (N14.InfoData.State=8 OR (Discrete_In.Input_Node_Count<15))
		AND (N15.InfoData.State=8 OR (Discrete_In.Input_Node_Count<16))
		AND (N16.InfoData.State=8 OR (Discrete_In.Input_Node_Count<17))
		AND (N17.InfoData.State=8 OR (Discrete_In.Input_Node_Count<18))
		AND (N18.InfoData.State=8 OR (Discrete_In.Input_Node_Count<19))
		AND (N19.InfoData.State=8 OR (Discrete_In.Input_Node_Count<20))
		AND (N20.InfoData.State=8 OR (Discrete_In.Input_Node_Count<21))
		AND (N21.InfoData.State=8 OR (Discrete_In.Input_Node_Count<22))
		AND (N22.InfoData.State=8 OR (Discrete_In.Input_Node_Count<23))
		AND (N100_STAT.InfoData.State=8 OR (Discrete_In.VB_Node_Count<1))
		AND (N101_STAT.InfoData.State=8 OR (Discrete_In.VB_Node_Count<2))
		AND (N102_STAT.InfoData.State=8 OR (Discrete_In.VB_Node_Count<3))

		THEN
			DiscreteNode_OK:=TRUE;

	ELSE
			DiscreteNode_OK:=FALSE;

	END_IF;



	(*Cable Break Detection*)
	(*Function Returns Flags to warn of possible cable break*)
	ECatSlave_Cable_Breaks:= FUN_GTAC_EcatSlaveConnState_64bit(NodeState);	























(*end*)
END_ACTION

ACTION Production:
(*$$$$$$$$$$$$$$$$$$$$$$$$$$$$$$$$$$$ Production Information $$$$$$$$$$$$$$$$$$$$$$$$$$$$$$$$$$$$$$$$$$*)
	(*Increment Production Counter*)
	Prod_Inc.CLK:= Unload_Complete;
	Prod_Inc();
	IF Prod_Inc.Q
		THEN
		Production_Count:= Production_Count+1;
	END_IF;
	IF Discrete_In.ResetProd
		THEN
		Production_Count:= 0;
	END_IF;
	Prod_Count_Out:= Production_Count;

(*~~~~~~~~~~~~~~~~~~~~~~~~~~~~~~~~Production Report~~~~~~~~~~~~~~~~~~~~~~~~~*)
	(*Input Data*)
	Production_Report.Machine_Serial:= GTAC_CONFIG.Machine_Serial;
	Production_Report.Machine_Common_Name:= GTAC_CONFIG.Machine_Common_Name;
	Production_Report.Prod_Inc:= Prod_Inc.Q;
	Production_Report.Scrap_Inc:= In_From_ICxx.QA_Request_RH;
	Production_Report.Scrap_Dec:= In_From_ICxx.QA_Reinsert_RH;
	Production_Report.Reference_TimeDate:= MAIN.Local_Time;
	Production_Report.Reference_Target_Time:= GTAC_CONFIG.ProdConfig_Target_CycleTime; 					(*This is the machine Expected Cycle Time*)
	Production_Report.Config_Day_TOD:= GTAC_CONFIG.ProdConfig_Day;										(*Pass Each Shift Configuration Structure (Start/End Time, Break Times etc*)
	Production_Report.Config_Aft_TOD:= GTAC_CONFIG.ProdConfig_Aft;
	Production_Report.Config_Mid_TOD:= GTAC_CONFIG.ProdConfig_Mid;
	Production_Report.Config_Shift_Enables:= GTAC_CONFIG.ProdConfig_Common.Shift_Enables;					(*Enable Bits for Shifts*)
	Production_Report.Config_Break_Count:= GTAC_CONFIG.ProdConfig_Common.Break_Count;						(*Select Amount of Breaks per shift*)
	Production_Report.Machine_StoppedBy_Fault:= Faults.System_Major_Fault;
	Production_Report.Enable_InShift_Change:= GTAC_CONFIG.ProdConfig_Option_SelectInShiftChange;				(*Allows Operator 5 mins at start and end of shift for clean up*)
	(*Call FB*)
	IF NOT MAIN.Starting_Scan_Pulse
		THEN
		Production_Report();
	END_IF;

(*~~~~~~~~~~~~~~~~~~~~~~~~~~~~~~~~ Cycle Time Counters ~~~~~~~~~~~~~~~~~~~~~~~~~*)
	(*Move Previous To Register*)
	Cycle_Time_Pulse.CLK:= Unload_Complete;
	Cycle_Time_Pulse();
	IF Cycle_Time_Pulse.Q
		THEN
		PrevCycle_Time_Out:= Cycle_Time_Out;
	END_IF;
	(*Monitor Current Cycle Time (Full Cycle Time of Process)*)
		Cycle_Time.PT:= T#9999S;
		Cycle_Time.IN:= NOT Cycle_Time_Pulse.Q AND In_Auto;
		Cycle_Time();
		Cycle_Time_Out:= Cycle_Time.ET;

	(*Monitor Load Time*)
		IF In_Auto AND NOT Start_Seal_Robots AND NOT Start_Stud_Robots AND NOT Start_Weld_Robots  AND NOT Weld_Robots_Clear AND NOT Unload_Complete
			THEN
			Load_Time_Out:= Load_Time.ET;
		END_IF;
		Load_Time.PT:= T#9999S;
		Load_Time.IN:= In_Auto AND NOT Start_Seal_Robots AND NOT Start_Stud_Robots AND NOT Start_Weld_Robots  AND NOT Weld_Robots_Clear AND NOT Unload_Complete;
		Load_Time();

	(*Monitor Robot Sealing Time*)
		IF NOT Seal_Robots_Clear
			THEN
			Seal_Time_Out:= Seal_Time.ET;
		END_IF;
		Seal_Time.PT:= T#9999S;
		Seal_Time.IN:= NOT Seal_Robots_Clear;
		Seal_Time();

	(*Monitor Robot Stud Time*)
		IF NOT Stud_Robots_Clear
			THEN
			Stud_Time_Out:= Stud_Time.ET;
		END_IF;
		Stud_Time.PT:= T#9999S;
		Stud_Time.IN:= NOT Stud_Robots_Clear;
		Stud_Time();

	(*Monitor Robot Welding Time*)
		IF NOT Weld_Robots_Clear
			THEN
			Weld_Time_Out:= Weld_Time.ET;
		END_IF;
		Weld_Time.PT:= T#9999S;
		Weld_Time.IN:= NOT Weld_Robots_Clear;
		Weld_Time();

	(*Monitor Robot Turntable Time*)
		IF NOT Turntable_Clear
			THEN
			Turn_Time_Out:= Turn_Time.ET;
		END_IF;
		Turn_Time.PT:= T#9999S;
		Turn_Time.IN:= NOT Turntable_Clear;
		Turn_Time();

	(*Monitor Unload Time*)
		IF Welding_Complete
			THEN
			Unload_Time_Out:= Unload_Time.ET;
		END_IF;
		Unload_Time.PT:= T#9999S;
		Unload_Time.IN:= Welding_Complete;
		Unload_Time();







(*~~~~~~~~~~~~~~~~~~~~~~~~~~~~~~~~Product Data Report~~~~~~~~~~~~~~~~~~~~~~~~~*)
(*Can be used to load and store product specific data (pass fail results, measurements etc) into DB*)
(*Triggers to start actual storage are contained in GTAC_CONFIG.Reports*)

(*Load Data into area*)
	Out_To_ICxx.ProductReport[24].Machine_Serial:= GTAC_CONFIG.Machine_Serial;
	Out_To_ICxx.ProductReport[24].Machine_Common_Name:= GTAC_CONFIG.Machine_Common_Name;
	Out_To_ICxx.ProductReport[24].Operator_ID:= 0;				(*for future*)
	Out_To_ICxx.ProductReport[24].Product_Serial:= 'Add product serial here';
	Out_To_ICxx.ProductReport[24].Product_Number:= 'Add product part number here';
	Out_To_ICxx.ProductReport[24].Product_Common_Name:= 'Add product common name here';
		(*Build part specific data arrays, simply leave un-used elements blank (Arrays are [0..31]*)
		(*Pass / Fail Notes - Used to capture overall terms like 'Pass' 'Fail' 'NA' etc.*)	
		Out_To_ICxx.ProductReport[24].Generic_PassFail_Notes[0]:= 'Fail';
		Out_To_ICxx.ProductReport[24].Generic_PassFail_Notes[1]:= 'Fail';
		
		(*Measurement Data - Used to capture specific measurment data*)	
		Out_To_ICxx.ProductReport[24].Generic_Measurements[0]:= 1.23450;
		Out_To_ICxx.ProductReport[24].Generic_Measurements[1]:= 0.54321;
END_ACTION

ACTION Proxies:


(*+++++++++++THIS AREA IS CUSTOM PER INSTALLATION AND WILL HAVE TO BE MODIFIED PER +++++++++++++*)
(*+++++++++++THIS AREA IS CUSTOM PER INSTALLATION AND WILL HAVE TO BE MODIFIED PER +++++++++++++*)



	(*Part 1 Present*)
		Part_Present1FB(
			Sensor_Input:= N01.I.0,
			On_Trigger1:= Enable_Motion AND In_Auto AND NOT Unload_Complete,
			On_Trigger2:= TRUE,
			Off_Trigger1:= Dry_Cycle OR (Cycle_Complete AND NOT Enable_Motion),
			Off_Trigger2:= TRUE,
			Disable_Faults:= FALSE,
			Fault_Delay:= T#1.5s,
			Status=> Part_Present1,
			Faulted=>  PPFaults.1);

	(*Part 2 Present*)
		Part_Present2FB(
			Sensor_Input:= N01.I.1,
			On_Trigger1:= Enable_Motion AND In_Auto AND NOT Unload_Complete,
			On_Trigger2:= TRUE,
			Off_Trigger1:= Dry_Cycle OR (Cycle_Complete  AND NOT Enable_Motion),
			Off_Trigger2:= TRUE,
			Disable_Faults:= FALSE,
			Fault_Delay:= T#1.5s,
			Status=> Part_Present2,
			Faulted=>  PPFaults.2);

	(*Part 3 Present*)
		Part_Present3FB(
			Sensor_Input:= N01.I.2,
			On_Trigger1:= Enable_Motion AND In_Auto AND NOT Unload_Complete,
			On_Trigger2:= TRUE,
			Off_Trigger1:= Dry_Cycle OR (Cycle_Complete  AND NOT Enable_Motion),
			Off_Trigger2:= TRUE,
			Disable_Faults:= FALSE,
			Fault_Delay:= T#1.5s,
			Status=> Part_Present3,
			Faulted=>  PPFaults.3);

	(*Part 4 Present*)
		Part_Present4FB(
			Sensor_Input:=N01.I.3,
			On_Trigger1:= Enable_Motion AND In_Auto AND NOT Unload_Complete,
			On_Trigger2:= TRUE,
			Off_Trigger1:= Dry_Cycle OR (Cycle_Complete  AND NOT Enable_Motion),
			Off_Trigger2:= TRUE,
			Disable_Faults:= FALSE,
			Fault_Delay:= T#1.5s,
			Status=> Part_Present4,
			Faulted=>  PPFaults.4);

	(*Part 5 Present*)
		Part_Present5FB(
			Sensor_Input:= N01.I.4,
			On_Trigger1:= Enable_Motion AND In_Auto AND NOT Unload_Complete,
			On_Trigger2:= TRUE,
			Off_Trigger1:= Dry_Cycle OR (Cycle_Complete  AND NOT Enable_Motion),
			Off_Trigger2:= TRUE,
			Disable_Faults:= FALSE,
			Fault_Delay:= T#1.5s,
			Status=> Part_Present5,
			Faulted=>  PPFaults.5);

	(*Part 6 Present*)
		Part_Present6FB(
			Sensor_Input:= N01.I.5,
			On_Trigger1:= Enable_Motion AND In_Auto AND NOT Unload_Complete,
			On_Trigger2:= TRUE,
			Off_Trigger1:= Dry_Cycle OR (Cycle_Complete  AND NOT Enable_Motion),
			Off_Trigger2:= TRUE,
			Disable_Faults:= FALSE,
			Fault_Delay:= T#1.5s,
			Status=> Part_Present6,
			Faulted=>  PPFaults.6);

	(*Part 7 Present*)
		Part_Present7FB(
			Sensor_Input:= N01.I.6,
			On_Trigger1:= Enable_Motion AND In_Auto AND NOT Unload_Complete,
			On_Trigger2:= TRUE,
			Off_Trigger1:= Dry_Cycle OR (Cycle_Complete  AND NOT Enable_Motion),
			Off_Trigger2:= TRUE,
			Disable_Faults:= FALSE,
			Fault_Delay:= T#1.5s,
			Status=> Part_Present7,
			Faulted=>  PPFaults.7);

	(*Part 8 Present*)
		Part_Present8FB(
			Sensor_Input:= N01.I.7,
			On_Trigger1:= Enable_Motion AND In_Auto AND NOT Unload_Complete,
			On_Trigger2:= TRUE,
			Off_Trigger1:= Dry_Cycle OR (Cycle_Complete  AND NOT Enable_Motion),
			Off_Trigger2:= TRUE,
			Disable_Faults:= FALSE,
			Fault_Delay:= T#1.5s,
			Status=> Part_Present8,
			Faulted=>  PPFaults.8);

	(*Part 9 Present*)
		Part_Present9FB(
			Sensor_Input:= N05.I.0,
			On_Trigger1:= Enable_Motion AND In_Auto AND NOT Unload_Complete,
			On_Trigger2:= TRUE,
			Off_Trigger1:= Dry_Cycle OR (Cycle_Complete  AND NOT Enable_Motion),
			Off_Trigger2:= TRUE,
			Disable_Faults:= FALSE,
			Fault_Delay:= T#1.5s,
			Status=> Part_Present9,
			Faulted=>  PPFaults.9);

	(*Part 10 Present*)
		Part_Present10FB(
			Sensor_Input:= N05.I.1,
			On_Trigger1:= Enable_Motion AND In_Auto AND NOT Unload_Complete,
			On_Trigger2:= TRUE,
			Off_Trigger1:= Dry_Cycle OR (Cycle_Complete  AND NOT Enable_Motion),
			Off_Trigger2:= TRUE,
			Disable_Faults:= FALSE,
			Fault_Delay:= T#1.5s,
			Status=> Part_Present10,
			Faulted=>  PPFaults.10);

	(*Part 11 Present*)
		Part_Present11FB(
			Sensor_Input:= N05.I.2,
			On_Trigger1:= Enable_Motion AND In_Auto AND NOT Unload_Complete,
			On_Trigger2:= TRUE,
			Off_Trigger1:= Dry_Cycle OR (Cycle_Complete  AND NOT Enable_Motion),
			Off_Trigger2:= TRUE,
			Disable_Faults:= FALSE,
			Fault_Delay:= T#1.5s,
			Status=> Part_Present11,
			Faulted=>  PPFaults.11);

	(*Part 12 Present*)
		Part_Present12FB(
			Sensor_Input:=  N05.I.3,
			On_Trigger1:= Enable_Motion AND In_Auto AND NOT Unload_Complete,
			On_Trigger2:= TRUE,
			Off_Trigger1:= Dry_Cycle OR (Cycle_Complete  AND NOT Enable_Motion),
			Off_Trigger2:= TRUE,
			Disable_Faults:= FALSE,
			Fault_Delay:= T#1.5s,
			Status=> Part_Present12,
			Faulted=>  PPFaults.12);

	(*Part 13 Present*)
		Part_Present13FB(
			Sensor_Input:= N05.I.4,
			On_Trigger1:= Enable_Motion AND In_Auto AND NOT Unload_Complete,
			On_Trigger2:= TRUE,
			Off_Trigger1:= Dry_Cycle OR (Cycle_Complete  AND NOT Enable_Motion),
			Off_Trigger2:= TRUE,
			Disable_Faults:= FALSE,
			Fault_Delay:= T#1.5s,
			Status=> Part_Present13,
			Faulted=>  PPFaults.13);

	(*Part 14 Present*)
		Part_Present14FB(
			Sensor_Input:= N05.I.5,
			On_Trigger1:= Enable_Motion AND In_Auto AND NOT Unload_Complete,
			On_Trigger2:= TRUE,
			Off_Trigger1:= Dry_Cycle OR (Cycle_Complete  AND NOT Enable_Motion),
			Off_Trigger2:= TRUE,
			Disable_Faults:= FALSE,
			Fault_Delay:= T#1.5s,
			Status=> Part_Present14,
			Faulted=>  PPFaults.14);


	(*Part 15 Present*)
		Part_Present15FB(
			Sensor_Input:= N05.I.6,
			On_Trigger1:= Enable_Motion AND In_Auto AND NOT Unload_Complete,
			On_Trigger2:= TRUE,
			Off_Trigger1:= Dry_Cycle OR (Cycle_Complete  AND NOT Enable_Motion),
			Off_Trigger2:= TRUE,
			Disable_Faults:= FALSE,
			Fault_Delay:= T#1.5s,
			Status=> Part_Present15,
			Faulted=>  PPFaults.15);

	(*Part 16 Present*)
		Part_Present16FB(
			Sensor_Input:= N05.I.7,
			On_Trigger1:= Enable_Motion AND In_Auto AND NOT Unload_Complete,
			On_Trigger2:= TRUE,
			Off_Trigger1:= Dry_Cycle OR (Cycle_Complete  AND NOT Enable_Motion),
			Off_Trigger2:= TRUE,
			Disable_Faults:= FALSE,
			Fault_Delay:= T#1.5s,
			Status=> Part_Present16,
			Faulted=>  PPFaults.16);

	(*Part 17 Present*)
		Part_Present17FB(
			Sensor_Input:= N06.I.0,
			On_Trigger1:= Enable_Motion AND In_Auto AND NOT Unload_Complete,
			On_Trigger2:= TRUE,
			Off_Trigger1:= Dry_Cycle OR (Cycle_Complete  AND NOT Enable_Motion),
			Off_Trigger2:= TRUE,
			Disable_Faults:= FALSE,
			Fault_Delay:= T#1.5s,
			Status=> Part_Present17,
			Faulted=>  PPFaults.17);

	(*Part 18 Present*)
		Part_Present18FB(
			Sensor_Input:= N06.I.1,
			On_Trigger1:= Enable_Motion AND In_Auto AND NOT Unload_Complete,
			On_Trigger2:= TRUE,
			Off_Trigger1:= Dry_Cycle OR (Cycle_Complete  AND NOT Enable_Motion),
			Off_Trigger2:= TRUE,
			Disable_Faults:= FALSE,
			Fault_Delay:= T#1.5s,
			Status=> Part_Present18,
			Faulted=>  PPFaults.18);

	(*Part 19 Present*)
		Part_Present19FB(
			Sensor_Input:= N06.I.2,
			On_Trigger1:= Enable_Motion AND In_Auto AND NOT Unload_Complete,
			On_Trigger2:= TRUE,
			Off_Trigger1:= Dry_Cycle OR (Cycle_Complete  AND NOT Enable_Motion),
			Off_Trigger2:= TRUE,
			Disable_Faults:= FALSE,
			Fault_Delay:= T#1.5s,
			Status=> Part_Present19,
			Faulted=>  PPFaults.19);

	(*Part 20 Present*)
		Part_Present20FB(
			Sensor_Input:= N06.I.3,
			On_Trigger1:= Enable_Motion AND In_Auto AND NOT Unload_Complete,
			On_Trigger2:= TRUE,
			Off_Trigger1:= Dry_Cycle OR (Cycle_Complete  AND NOT Enable_Motion),
			Off_Trigger2:= TRUE,
			Disable_Faults:= FALSE,
			Fault_Delay:= T#1.5s,
			Status=> Part_Present20,
			Faulted=>  PPFaults.20);

	(*Part 21 Present*)
		Part_Present21FB(
			Sensor_Input:= N06.I.4,
			On_Trigger1:= Enable_Motion AND In_Auto AND NOT Unload_Complete,
			On_Trigger2:= TRUE,
			Off_Trigger1:= Dry_Cycle OR (Cycle_Complete  AND NOT Enable_Motion),
			Off_Trigger2:= TRUE,
			Disable_Faults:= FALSE,
			Fault_Delay:= T#1.5s,
			Status=> Part_Present21,
			Faulted=>  PPFaults.21);

	(*Part 22 Present*)
		Part_Present22FB(
			Sensor_Input:= N06.I.5,
			On_Trigger1:= Enable_Motion AND In_Auto AND NOT Unload_Complete,
			On_Trigger2:= TRUE,
			Off_Trigger1:= Dry_Cycle OR (Cycle_Complete  AND NOT Enable_Motion),
			Off_Trigger2:= TRUE,
			Disable_Faults:= FALSE,
			Fault_Delay:= T#1.5s,
			Status=> Part_Present22,
			Faulted=>  PPFaults.22);

	(*Part 23 Present*)
		Part_Present23FB(
			Sensor_Input:= N06.I.6,
			On_Trigger1:= Enable_Motion AND In_Auto AND NOT Unload_Complete,
			On_Trigger2:= TRUE,
			Off_Trigger1:= Dry_Cycle OR (Cycle_Complete  AND NOT Enable_Motion),
			Off_Trigger2:= TRUE,
			Disable_Faults:= FALSE,
			Fault_Delay:= T#1.5s,
			Status=> Part_Present23,
			Faulted=>  PPFaults.23);

	(*Part 24 Present*)
		Part_Present24FB(
			Sensor_Input:= N06.I.7,
			On_Trigger1:= Enable_Motion AND In_Auto AND NOT Unload_Complete,
			On_Trigger2:= TRUE,
			Off_Trigger1:= Dry_Cycle OR (Cycle_Complete  AND NOT Enable_Motion),
			Off_Trigger2:= TRUE,
			Disable_Faults:= FALSE,
			Fault_Delay:= T#1.5s,
			Status=> Part_Present24,
			Faulted=>  PPFaults.24);

	(*Part 25 Present*)
		Part_Present25FB(
			Sensor_Input:= N07.I.0,
			On_Trigger1:= Enable_Motion AND In_Auto AND NOT Unload_Complete,
			On_Trigger2:= TRUE,
			Off_Trigger1:= Dry_Cycle OR (Cycle_Complete  AND NOT Enable_Motion),
			Off_Trigger2:= TRUE,
			Disable_Faults:= FALSE,
			Fault_Delay:= T#1.5s,
			Status=> Part_Present25,
			Faulted=>  PPFaults.25);

	(*Part 26 Present*)
		Part_Present26FB(
			Sensor_Input:= N07.I.1,
			On_Trigger1:= Enable_Motion AND In_Auto AND NOT Unload_Complete,
			On_Trigger2:= TRUE,
			Off_Trigger1:= Dry_Cycle OR (Cycle_Complete  AND NOT Enable_Motion),
			Off_Trigger2:= TRUE,
			Disable_Faults:= FALSE,
			Fault_Delay:= T#1.5s,
			Status=> Part_Present26,
			Faulted=>  PPFaults.26);

	(*Part 27 Present*)
		Part_Present27FB(
			Sensor_Input:= N07.I.2,
			On_Trigger1:= Enable_Motion AND In_Auto AND NOT Unload_Complete,
			On_Trigger2:= TRUE,
			Off_Trigger1:= Dry_Cycle OR (Cycle_Complete  AND NOT Enable_Motion),
			Off_Trigger2:= TRUE,
			Disable_Faults:= FALSE,
			Status=> Part_Present27,
			Faulted=>  PPFaults.27);

	(*Part 28 Present*)
		Part_Present28FB(
			Sensor_Input:= N07.I.3,
			On_Trigger1:= Enable_Motion AND In_Auto AND NOT Unload_Complete,
			On_Trigger2:= TRUE,
			Off_Trigger1:= Dry_Cycle OR (Cycle_Complete  AND NOT Enable_Motion),
			Off_Trigger2:= TRUE,
			Disable_Faults:= FALSE,
			Fault_Delay:= T#1.5s,
			Status=> Part_Present28,
			Faulted=>  PPFaults.28);


	(*Part 29 Present*)
		Part_Present29FB(
			Sensor_Input:= N07.I.4,
			On_Trigger1:= Enable_Motion AND In_Auto AND NOT Unload_Complete,
			On_Trigger2:= TRUE,
			Off_Trigger1:= Dry_Cycle OR (Cycle_Complete  AND NOT Enable_Motion),
			Off_Trigger2:= TRUE,
			Disable_Faults:= FALSE,
			Fault_Delay:= T#1.5s,
			Status=> Part_Present29,
			Faulted=>  PPFaults1.0);

	(*Part 30 Present*)
		Part_Present30FB(
			Sensor_Input:=N07.I.5,
			On_Trigger1:= Enable_Motion AND In_Auto AND NOT Unload_Complete,
			On_Trigger2:= TRUE,
			Off_Trigger1:= Dry_Cycle OR (Cycle_Complete  AND NOT Enable_Motion),
			Off_Trigger2:= TRUE,
			Disable_Faults:= FALSE,
			Fault_Delay:= T#1.5s,
			Status=> Part_Present30,
			Faulted=>  PPFaults1.1);

	(*Part 31 Present*)
		Part_Present31FB(
			Sensor_Input:= N07.I.6,
			On_Trigger1:= Enable_Motion AND In_Auto AND NOT Unload_Complete,
			On_Trigger2:= TRUE,
			Off_Trigger1:= Dry_Cycle OR (Cycle_Complete  AND NOT Enable_Motion),
			Off_Trigger2:= TRUE,
			Disable_Faults:= FALSE,
			Fault_Delay:= T#1.5s,
			Status=> Part_Present31,
			Faulted=>  PPFaults1.2);

	(*Part 32 Present*)
		Part_Present32FB(
			Sensor_Input:= N07.I.7,
			On_Trigger1:= Enable_Motion AND In_Auto AND NOT Unload_Complete,
			On_Trigger2:= TRUE,
			Off_Trigger1:= Dry_Cycle OR (Cycle_Complete  AND NOT Enable_Motion),
			Off_Trigger2:= TRUE,
			Disable_Faults:= FALSE,
			Fault_Delay:= T#1.5s,
			Status=> Part_Present32,
			Faulted=>  PPFaults1.3);

	(*Part 33 Present*)
		Part_Present33FB(
			Sensor_Input:= N08.I.0,
			On_Trigger1:= Enable_Motion AND In_Auto AND NOT Unload_Complete,
			On_Trigger2:= TRUE,
			Off_Trigger1:= Dry_Cycle OR (Cycle_Complete  AND NOT Enable_Motion),
			Off_Trigger2:= TRUE,
			Disable_Faults:= FALSE,
			Fault_Delay:= T#1.5s,
			Status=> Part_Present33,
			Faulted=>  PPFaults1.4);

	(*Part 34 Present*)
		Part_Present34FB(
			Sensor_Input:= N08.I.1,
			On_Trigger1:= Enable_Motion AND In_Auto AND NOT Unload_Complete,
			On_Trigger2:= TRUE,
			Off_Trigger1:= Dry_Cycle OR (Cycle_Complete  AND NOT Enable_Motion),
			Off_Trigger2:= TRUE,
			Disable_Faults:= FALSE,
			Fault_Delay:= T#1.5s,
			Status=> Part_Present34,
			Faulted=>  PPFaults1.5);

	(*Part 35 Present*)
		Part_Present35FB(
			Sensor_Input:= N08.I.2,
			On_Trigger1:= Enable_Motion AND In_Auto AND NOT Unload_Complete,
			On_Trigger2:= TRUE,
			Off_Trigger1:= Dry_Cycle OR (Cycle_Complete  AND NOT Enable_Motion),
			Off_Trigger2:= TRUE,
			Disable_Faults:= FALSE,
			Fault_Delay:= T#1.5s,
			Status=> Part_Present35,
			Faulted=>  PPFaults1.6);

	(*Part 36 Present*)
		Part_Present36FB(
			Sensor_Input:= N08.I.3,
			On_Trigger1:= Enable_Motion AND In_Auto AND NOT Unload_Complete,
			On_Trigger2:= TRUE,
			Off_Trigger1:= Dry_Cycle OR (Cycle_Complete  AND NOT Enable_Motion),
			Off_Trigger2:= TRUE,
			Disable_Faults:= FALSE,
			Fault_Delay:= T#1.5s,
			Status=> Part_Present36,
			Faulted=>  PPFaults1.7);

	(*Part 37 Present*)
		Part_Present37FB(
			Sensor_Input:= N08.I.4,
			On_Trigger1:= Enable_Motion AND In_Auto AND NOT Unload_Complete,
			On_Trigger2:= TRUE,
			Off_Trigger1:= Dry_Cycle OR (Cycle_Complete  AND NOT Enable_Motion),
			Off_Trigger2:= TRUE,
			Disable_Faults:= FALSE,
			Fault_Delay:= T#1.5s,
			Status=> Part_Present37,
			Faulted=>  PPFaults1.8);

	(*Part 38 Present*)
		Part_Present38FB(
			Sensor_Input:= N08.I.5,
			On_Trigger1:= Enable_Motion AND In_Auto AND NOT Unload_Complete,
			On_Trigger2:= TRUE,
			Off_Trigger1:= Dry_Cycle OR (Cycle_Complete  AND NOT Enable_Motion),
			Off_Trigger2:= TRUE,
			Disable_Faults:= FALSE,
			Fault_Delay:= T#1.5s,
			Status=> Part_Present38,
			Faulted=>  PPFaults1.9);

	(*Part 39 Present*)
		Part_Present39FB(
			Sensor_Input:= N08.I.6,
			On_Trigger1:= Enable_Motion AND In_Auto AND NOT Unload_Complete,
			On_Trigger2:= TRUE,
			Off_Trigger1:= Dry_Cycle OR (Cycle_Complete  AND NOT Enable_Motion),
			Off_Trigger2:= TRUE,
			Disable_Faults:= FALSE,
			Fault_Delay:= T#1.5s,
			Status=> Part_Present39,
			Faulted=>  PPFaults1.10);

	(*Part 40 Present*)
		Part_Present40FB(
			Sensor_Input:= N08.I.7,
			On_Trigger1:= Enable_Motion AND In_Auto AND NOT Unload_Complete,
			On_Trigger2:= TRUE,
			Off_Trigger1:= Dry_Cycle OR (Cycle_Complete  AND NOT Enable_Motion),
			Off_Trigger2:= TRUE,
			Disable_Faults:= FALSE,
			Fault_Delay:= T#1.5s,
			Status=> Part_Present40,
			Faulted=>  PPFaults1.11);



(*end*)
END_ACTION

ACTION Robot_Registration:


(*#################################### Register Robots to Tool ##################################*)
(*+++++++++++THIS AREA IS CUSTOM PER INSTALLATION AND WILL HAVE TO BE MODIFIED PER +++++++++++++*)
(*+++++++++++THIS AREA IS CUSTOM PER INSTALLATION AND WILL HAVE TO BE MODIFIED PER +++++++++++++*)
(*NOTE: See Example code in Fix 15 / 16*)
(*NOTE: See Example code in Fix 15 / 16*)

	(*Data From Load Robot(s)*)
	Load_Robots_Clear1:= TRUE;
	Load_Robots_Clear2:= TRUE;
	Load_Robots_Clear:=Load_Robots_Clear1 AND Load_Robots_Clear2;
	Load_Robots_WorkingOK1:= FALSE;
	Load_Robots_WorkingOK2:= FALSE;
	IF FALSE
		THEN
		Load_Robots_UnclampEarly1:= TRUE;
	END_IF;
	IF FALSE
		THEN
		Load_Robots_UnclampEarly2:= TRUE;
	END_IF;
	Load_Robots_Complete1:= FALSE;
	Load_Robots_Complete2:= FALSE;
	Load_Robots_PartInEOAT1:= FALSE;
	Load_Robots_PartInEOAT2:= FALSE;


	(*Data From Turntable*)
	TurntableA_Clear:= TRUE;
	TurntableB_Clear:= TRUE;
	Turntable_Clear:= TurntableA_Clear AND TurntableB_Clear AND NOT MAIN.R1.In_Teach;
	TurntableA_At_Robot:= FALSE;
	TurntableB_At_Robot:= FALSE;
	Turntable_WorkingOK:= FALSE;
	TurntableA_Complete:= FALSE;
	TurntableB_Complete:= FALSE;


	(*Data From Seal Robot(s)*)
	Seal_Robots_Clear:= TRUE;
	Seal_Robots_WorkingOK:= FALSE;
	IF FALSE
		THEN
		Seal_Robots_UnclampEarly:= TRUE;
	END_IF;
	Seal_Robots_Complete:= FALSE;


	(*Data From Stud Robot(s)*)
	Stud_Robots_Clear:= TRUE;
	Stud_Robots_WorkingOK:= FALSE;
	IF FALSE
		THEN
		Stud_Robots_UnclampEarly:= TRUE;
	END_IF;
	Stud_Robots_Complete:= FALSE;


	(*Data From Weld Robot(s)*)
	Weld_Robots_Clear:= TRUE;
	Weld_Robots_WorkingOK:= FALSE;
	IF FALSE
		THEN
		Weld_Robots_UnclampEarly:= TRUE;
	END_IF;
	Weld_Robots_Complete:= FALSE;

	(*Change Robots for Current Fixture functionality*) (*If no MIG robots Set to True.  Example code is in Fix15/16*) 
	Mig_Robots_Ready:=	TRUE;
	
	(*Data From Unload Robot(s)*)
	Unload_Robots_Clear1:= TRUE;
	Unload_Robots_Clear2:= TRUE;
	Unload_Robots_Clear:= Unload_Robots_Clear1 AND Unload_Robots_Clear2;
	Unload_Robots_WorkingOK1:= FALSE;
	Unload_Robots_WorkingOK2:= FALSE;
	Unload_Robots_Complete1:= FALSE;
	Unload_Robots_Complete2:= FALSE;
	Unload_Robots_EOATEmpty1:=FALSE;
	Unload_Robots_EOATEmpty2:= FALSE;



	(*Amalgumate All Robots Clear of Tool*)
	All_Robots_Clear:= Load_Robots_Clear AND Seal_Robots_Clear AND Stud_Robots_Clear AND Turntable_Clear AND Weld_Robots_Clear AND Unload_Robots_Clear;

	(*Data To All Robots*)
	(*Task ID*)
	R1_Data.Task_ID[1]:=Task_ID;

	(*Fix ID*)
	R1_Data.Fix_ID[1]:=Fix_ID;

	(*Model ID*)
	R1_Data.Model_ID[1]:=Model_ID;

	(*Proceed from Pounce*)
	R1_Data.Proceed_From_Pounce[1]:= Robots_Clear_ToProceed;

	(*Complete Acks*)
	R1_Data.Complete_Ack[1]:=(Weld_Complete_Ack AND Weld_Robots_WorkingOK);

	(*Repo Acks*)
	R1_Data.PeripheralReq_Ack[1]:= Repo_Ack;

(*%%%%%%%%%%%%%% Call Robots to Tool and Give Them, Task ID, Fixture ID and Model ID %%%%%%%%%%%%%%%%%*)
	(* Perform Call To Tool*)
	Tool_Call_ForLoadRobots1:= Enable_Motion AND (NOT Cell_In_Services OR NOT Load_Robots_Clear1)
						AND Start_Load_Robots1 AND NOT Start_Load_Robots2 AND NOT Start_Weld_Robots AND NOT Start_Seal_Robots AND NOT Start_Stud_Robots
						AND NOT Start_Unload_Robots1 AND NOT Start_Unload_Robots2 AND NOT Start_TurntableA AND NOT Start_TurntableB;
	Tool_Call_ForLoadRobots2:= Enable_Motion AND (NOT Cell_In_Services OR NOT Load_Robots_Clear2)
						AND NOT Start_Load_Robots1 AND Start_Load_Robots2 AND NOT Start_Weld_Robots AND NOT Start_Seal_Robots AND NOT Start_Stud_Robots
						AND NOT Start_Unload_Robots1 AND NOT Start_Unload_Robots2 AND NOT Start_TurntableA AND NOT Start_TurntableB;
	Tool_Call_ForSealRobots:=Enable_Motion AND (NOT Cell_In_Services OR NOT Seal_Robots_Clear)
						AND NOT Start_Load_Robots1 AND NOT Start_Load_Robots2 AND NOT Start_Weld_Robots AND Start_Seal_Robots AND NOT Start_Stud_Robots
						AND NOT Start_Unload_Robots1 AND NOT Start_Unload_Robots2 AND NOT Start_TurntableA AND NOT Start_TurntableB;
	Tool_Call_ForStudRobots:=Enable_Motion AND (NOT Cell_In_Services OR NOT Stud_Robots_Clear)
						AND NOT Start_Load_Robots1 AND NOT Start_Load_Robots2 AND NOT Start_Weld_Robots AND NOT Start_Seal_Robots AND Start_Stud_Robots
						AND NOT Start_Unload_Robots1 AND NOT Start_Unload_Robots2 AND NOT Start_TurntableA AND NOT Start_TurntableB;
	Tool_Call_ForSweepA:= Enable_Motion AND (NOT Cell_In_Services OR NOT TurntableA_Clear)
						AND NOT Start_Load_Robots1 AND NOT Start_Load_Robots2 AND NOT Start_Weld_Robots AND NOT Start_Seal_Robots AND NOT Start_Stud_Robots
						AND NOT Start_Unload_Robots1 AND NOT Start_Unload_Robots2 AND Start_TurntableA AND NOT Start_TurntableB;
	Tool_Call_ForSweepB:= Enable_Motion AND (NOT Cell_In_Services OR NOT TurntableB_Clear)
						AND NOT Start_Load_Robots1 AND NOT Start_Load_Robots2 AND NOT Start_Weld_Robots AND NOT Start_Seal_Robots AND NOT Start_Stud_Robots
						AND NOT Start_Unload_Robots1 AND NOT Start_Unload_Robots2 AND NOT Start_TurntableA AND Start_TurntableB;
	Tool_Call_ForWeldRobots:= Enable_Motion AND (NOT Cell_In_Services OR NOT Weld_Robots_Clear)
						AND NOT Start_Load_Robots1 AND NOT Start_Load_Robots2 AND Start_Weld_Robots AND NOT Start_Seal_Robots AND NOT Start_Stud_Robots
						AND NOT Start_Unload_Robots1 AND NOT Start_Unload_Robots2 AND NOT Start_TurntableA AND NOT Start_TurntableB;
	Tool_Call_ForUnloadRobots1:= Enable_Motion AND (NOT Cell_In_Services OR NOT Unload_Robots_Clear1)
						AND NOT Start_Load_Robots1 AND NOT Start_Load_Robots2 AND NOT Start_Weld_Robots AND NOT Start_Seal_Robots AND NOT Start_Stud_Robots
						AND Start_Unload_Robots1 AND NOT Start_Unload_Robots2 AND NOT Start_TurntableA AND NOT Start_TurntableB;
	Tool_Call_ForUnloadRobots2:= Enable_Motion AND (NOT Cell_In_Services OR NOT Unload_Robots_Clear2)
						AND NOT Start_Load_Robots1 AND NOT Start_Load_Robots2 AND NOT Start_Weld_Robots AND NOT Start_Seal_Robots AND NOT Start_Stud_Robots
						AND NOT Start_Unload_Robots1 AND Start_Unload_Robots2 AND NOT Start_TurntableA AND NOT Start_TurntableB;



	(*Allow Robots to Proceed Into Tool*)
	(*!!!!!This is the final OK to allow Robots Into the Tool Area, So it Better Be Ready!!!!!!!*)
	IF Enable_Motion
		THEN
			IF Load_Robots_Proceed1 AND Load_Robots_WorkingOK1 AND Load_Robots_Clear2 AND Seal_Robots_Clear AND Stud_Robots_Clear AND Turntable_Clear AND Weld_Robots_Clear AND Unload_Robots_Clear
				THEN Robots_Clear_ToProceed:=TRUE;
			ELSIF Load_Robots_Proceed2 AND Load_Robots_WorkingOK2 AND Load_Robots_Clear1 AND Seal_Robots_Clear AND Stud_Robots_Clear AND Turntable_Clear AND Weld_Robots_Clear AND Unload_Robots_Clear
				THEN Robots_Clear_ToProceed:=TRUE;
			ELSIF Seal_Robots_Proceed AND Seal_Robots_WorkingOK AND Load_Robots_Clear AND Stud_Robots_Clear AND Turntable_Clear AND Weld_Robots_Clear AND Unload_Robots_Clear
				THEN Robots_Clear_ToProceed:=TRUE;
			ELSIF Stud_Robots_Proceed AND Stud_Robots_WorkingOK AND Load_Robots_Clear AND Seal_Robots_Clear AND Turntable_Clear AND Weld_Robots_Clear AND Unload_Robots_Clear
				THEN Robots_Clear_ToProceed:=TRUE;
			ELSIF Weld_Robots_Proceed AND Weld_Robots_WorkingOK AND Load_Robots_Clear AND Seal_Robots_Clear AND Stud_Robots_Clear AND Turntable_Clear AND Unload_Robots_Clear
				THEN Robots_Clear_ToProceed:=TRUE;
			ELSIF Unload_Robots_Proceed1 AND Unload_Robots_WorkingOK1 AND Load_Robots_Clear AND Seal_Robots_Clear AND Stud_Robots_Clear AND Turntable_Clear AND Weld_Robots_Clear AND Unload_Robots_Clear2
				THEN Robots_Clear_ToProceed:=TRUE;
			ELSIF Unload_Robots_Proceed2 AND Unload_Robots_WorkingOK2 AND Load_Robots_Clear AND Seal_Robots_Clear AND Stud_Robots_Clear AND Turntable_Clear AND Weld_Robots_Clear AND Unload_Robots_Clear1
				THEN Robots_Clear_ToProceed:=TRUE;
			ELSE Robots_Clear_ToProceed:= FALSE;
			END_IF;
		ELSE Robots_Clear_ToProceed:= FALSE;
	END_IF;

(*+++++++++++++++++++++++++++++++++++++++++++++++ Task Complete Acks ++++++++++++++++++++++++++*)
	(*1st Load Complete Ack*)
	Load_Complete1_Ack:= Load_Robots_Complete1 AND Load_Complete1;

	(*2nd Load Complete Ack*)
	Load_Complete2_Ack:= Load_Robots_Complete2 AND Load_Complete2;

	(*Seal Complete Ack*)
	Seal_Complete_Ack:= Seal_Robots_Complete AND Sealing_Complete;

	(*Stud Complete Ack*)
	Stud_Complete_Ack:= Stud_Robots_Complete AND Stud_Complete;

	(*Sweep Complete ACK*)
	TurnA_Complete_Ack := TurntableA_Complete AND TurntableA_At_Robot;
	TurnB_Complete_Ack := TurntableB_Complete AND TurntableB_At_Robot;

	(*Weld Complete Ack*)
	Weld_Complete_Ack:= Weld_Robots_Complete AND Welding_Complete;

	(*Unload Complete Ack*)
	Unload_Complete1_Ack:= Unload_Robots_Complete1 AND Unload_Complete;

	(*Unload Complete Ack*)
	Unload_Complete2_Ack:= Unload_Robots_Complete2 AND Unload_Complete;




(*end*)
END_ACTION

ACTION Status_and_Faults:



